	m_stabilizerDeployedFlag : BOOL;
	
	m_sdrivingLeverSensorManualFlag : BOOL;
	
	m_trocarOnFlag :INT;

	m_uiControl : ST_uiControl;
	
	m_joystickValue : vec8d;
	
	m_jntPosReachLimit : vec8b;
	
	m_inMotion : BOOL := false;
END_STRUCT
END_TYPE

// ---- DUTs/Structure/TasksCommunication/ST_CartUIData.TcDUT
TYPE ST_CartUIData :
STRUCT
	m_joystickDataFromUI:ARRAY [0..21] OF USINT;
	m_ctrlEnableFromUI:ST_uiControl;
	m_standColumnHightLimit :LREAL;
	m_surgicalSite : UINT;
	m_surgicalLocation : UINT;
	m_cartDrapingState : UINT;
	m_cartDockingState : UINT;
	m_cartSpecificPosDocking : Vec8d;
	m_cartSpecificPosDraping : Vec8d;
END_STRUCT
END_TYPE

// ---- DUTs/Structure/TasksCommunication/ST_SetupStatus.TcDUT
TYPE ST_SetupStatus :
STRUCT
	// state machine
	m_armState:ARRAY[1..g_sArmNum] OF E_SetupArmState:=[g_sArmNum(SetupArmState_Error)];
	
	// current pose of set arm distal end
	m_curEndPose:ARRAY[1..g_sArmNum] OF ST_Frame;
	
	// position of remote center point
	m_rcPos :ARRAY[1..g_sArmNum] OF Vec3d;
END_STRUCT
END_TYPE

// ---- DUTs/Structure/TasksCommunication/ST_SetupJointData.TcDUT
TYPE ST_SetupJointData :
STRUCT
	// joint position compute with motor encoder
	m_curMotorPos :ARRAY[1..g_sArmNum] OF Vec5d;
	
	// joint position compute with link/abs encoder
	m_curLinkPos :ARRAY[1..g_sArmNum] OF Vec5d;
	
	// target joint position 
	m_cmdJntPos :ARRAY[1..g_sArmNum] OF Vec5d;
	
	// current joint position 
	m_curJntPos :ARRAY[1..g_sArmNum] OF Vec5d;
	
	// current joint position 
	m_curJntVel :ARRAY[1..g_sArmNum] OF Vec5d;
	
	// raw joint current  
	m_rawJntCurrent :ARRAY[1..g_sArmNum] OF Vec5d;
	
	// command joint current 
	m_cmdJntCurrent :ARRAY[1..g_sArmNum] OF Vec5d;
	
END_STRUCT
END_TYPE

// ---- DUTs/Structure/TasksCommunication/ST_SlaveDynaData.TcDUT
TYPE ST_SlaveDynaData :
STRUCT
	// mass matrix in joint space
	m_massMat :ARRAY[1..g_sArmNum] OF Mat3d;
	
	// gravity
	m_gravity :ARRAY[1..g_sArmNum] OF Vec3d;
	
	// instrument out-of-view data
	m_insruViewData :ARRAY[1..g_sArmNum] OF Vec3i;
END_STRUCT
END_TYPE

// ---- DUTs/Structure/TasksCommunication/ST_SlaveUIData.TcDUT
// Output from UI controller
// Input to slave arm control task and cart control task  
TYPE ST_SlaveUIData :
STRUCT
	m_slaveArmDisableFlag :ARRAY[1..4] OF BOOL:=[4(FALSE)];
	m_instruUsageWrite :ARRAY[1..4] OF BOOL:=[4(FALSE)];
	m_armInSelfCheck :  ARRAY [1..g_sArmNum] OF BOOL;
	m_armSelfCheckFinshed :  ARRAY [1..g_sArmNum] OF BOOL;
	m_dumpEnergy : UINT:=51;
END_STRUCT
END_TYPE

// ---- DUTs/Structure/TasksCommunication/ST_MasterJointData.TcDUT
// Output from master arm control task 
// Input to safety task and force controller task
TYPE ST_MasterJointData :
STRUCT
	// joint position compute with motor encoder
	m_curMotorPos :ARRAY[1..g_mArmNum] OF Vec7d;
	
	// joint position compute with link/abs encoder
	m_curLinkPos :ARRAY[1..g_mArmNum] OF Vec7d;
	
	// target joint position 
	m_cmdJntPos :ARRAY[1..g_mArmNum] OF Vec7d;
	
	// current joint position 
	m_curJntPos :ARRAY[1..g_mArmNum] OF Vec7d;
	
	// target joint velocity 
	m_cmdJntVel :ARRAY[1..g_mArmNum] OF Vec7d;
	
	// current joint position 
	m_curJntVel :ARRAY[1..g_mArmNum] OF Vec7d;
	
	// command joint torque 
	m_cmdJntTrq :ARRAY[1..g_mArmNum] OF Vec7d;
	
	// current joint torque 
	m_curJntTrq :ARRAY[1..g_mArmNum] OF Vec7d;
	
	// raw joint current  
	m_rawJntCurrent :ARRAY[1..g_mArmNum] OF Vec7d;
	
	// filtd  joint current  
	m_filtJntCurrent :ARRAY[1..g_mArmNum] OF Vec7d;
	
END_STRUCT
END_TYPE

// ---- DUTs/Structure/TasksCommunication/ST_MotorInputs.TcDUT
TYPE ST_MotorInputs:
STRUCT
	// driver error info
	m_driverError:UDINT;
	
	// driver ethercat status
	m_statusWord:UINT;
	
	// motor/relative encoder from IO
	m_motorEncoder :DINT;
	
	// link/absolute encoder form IO
	m_linkEncoder :DINT;
	
	// motor current from IO
	m_current : DINT;
	
	//motor electrical angle deviation
	m_electriAngleDev : DINT;
	
END_STRUCT
END_TYPE

// ---- DUTs/Structure/TasksCommunication/ST_MotorOutputs.TcDUT
TYPE ST_MotorOutputs :
STRUCT
	// driver control word
	m_controlWord: UINT :=DriverCtrlWord_INIT;
	
	// motor control mode, 0 for position mode, 1 for torque mode
	m_opMode : SINT :=INT_TO_SINT(DriverOPMode_Pos);;
	
	// target motor encoder
	m_cmdMotorEncoder :DINT := 0;
	
	// motor current to IO
	m_cmdCurrent :DINT := 0;
	
	//Powerbox rated current
	m_ratedCurrent:DINT;
END_STRUCT
END_TYPE

// ---- DUTs/Structure/TasksCommunication/ST_SlaveJointData.TcDUT
TYPE ST_SlaveJointData :
STRUCT
	
	// joint position compute with motor encoder
	m_curMotorPos :ARRAY[1..g_sArmNum] OF Vec8d;
	
	// joint position compute with link/abs encoder
	m_curLinkPos :ARRAY[1..g_sArmNum] OF Vec8d;
	
	// target joint position 
	m_cmdJntPos :ARRAY[1..g_sArmNum] OF Vec8d;
	
	// current joint position 
	m_curJntPos :ARRAY[1..g_sArmNum] OF Vec8d;
	
	// current joint position 
	m_curJntVel :ARRAY[1..g_sArmNum] OF Vec8d;
	
	// raw joint current  
	m_rawJntCurrent :ARRAY[1..g_sArmNum] OF Vec8d;
	
	// command joint current 
	m_cmdJntCurrent :ARRAY[1..g_sArmNum] OF Vec8d;
	
	// slave DH joint position 
	m_curDHJntPos :ARRAY[1..g_sArmNum] OF Vec6d;
END_STRUCT
END_TYPE

// ---- DUTs/Structure/TasksCommunication/ST_SafetyData.TcDUT
// Output from safety check task
// Input to master arm control task
TYPE ST_SafetyData :
STRUCT
	m_slaveErrFlag :ARRAY[1..g_sArmNum] OF BOOL :=[4(FALSE)];
	m_setupErrFlag :ARRAY[1..g_sArmNum] OF BOOL :=[4(FALSE)];
	m_cartErrFlag :BOOL :=FALSE;
	m_cartSteadyFootErr :BOOL;
	m_cartWheelErr :BOOL;
	m_cartStandColumnErr :BOOL;
	m_cartAdjustErr :BOOL;
	m_cartOverhangErr :BOOL;
END_STRUCT
END_TYPE

// ---- DUTs/Structure/ST_SlaveArmCtrlCmds.TcDUT
TYPE ST_SlaveArmCtrlCmds :
STRUCT
	// arm control data
	// NOTE: simulated joint position is usd for kinematic controller 
	//		while command joint position is used for real robot controller
	// 		They are identical for the most time, but in some cases, simulated position is filted to get command one 
	m_jntEnableFlag : Vec8i;
	m_jntOPMode : Vec8i;
	m_simJntPos : Vec8d;
	m_cmdJntPos : VEC8d;
	m_cmdJntVel : VEC8d;
	m_cmdJntAcc : VEC8d:=g_zeroVec8d;
	m_cmdJntTrq : VEC8d:=g_zeroVec8d;
	m_cmdCartPose : ST_Frame;
	m_cmdCartTwist : Vec6d;
	m_FFJntTrq :Vec8d:=g_zeroVec8d;
	m_stiffFlag:Vec8i; //---1028
END_STRUCT
END_TYPE

// ---- DUTs/Structure/ST_SlaveInputDataPool.TcDUT
// Struct contains all data from other tasks and controller used for slave control
TYPE ST_SlaveInputDataPool :
STRUCT
		
	// UI information, import from UI controller
	m_UIData :ST_SlaveUIData;
	
	// safety information, import from safety check task
	m_safetyData AT %I*: ST_SafetyData;
	
	// master robot status, copy from MSCommu_MasterStatus
	m_masterStatus :ST_MasterStatus;
	
	// setup arms infromation;
	m_setupStatus AT %I* : ST_SetupStatus;
	
	// slave dynamic data
	m_slaveDynaData AT %I* : ST_SlaveDynaData;
	
END_STRUCT
END_TYPE

// ---- DUTs/Structure/UICommunication/ST_cartOperation.TcDUT
TYPE ST_cartOperation :
STRUCT
	//sterile state ,  0 : unfinshed  , 1 : complete
	m_setupSterileStateArm1 : UINT;
	m_setupSterileStateArm2 : UINT;
	m_setupSterileStateArm3 : UINT;
	m_setupSterileStateArm4 : UINT;
	
	//draping adjust state , 0 : unfinshed  , 1 : finshed
	m_drapingAdjustState : UINT;

	//sterile install state , 0 : unfinshed  , 1 : finshed
	m_setupSterileState : UINT;

	//docking adjust state , 0 : unfinshed  , 1 : finshed
	m_dockingAdjustState : UINT;
	
	//cart in the sterile area 
	m_cartInSterileState : UINT;
	
	//scope installed , 0 : unfinshed  , 1 : finshed
	m_scopeInstalled :UINT;
	
	//robot in surgical allowed , scope installed and an arm mounted instrument
	m_inSurgicalAllowed : UINT;
	
	//arm storage completed
	m_armStorageCompleted : UINT;
END_STRUCT
END_TYPE

// ---- DUTs/Structure/UICommunication/ST_instruInfomation.TcDUT
TYPE ST_instruInfomation :
STRUCT
	//instrument is ready
	m_instruIsConnected : BOOL;
	
	//new instrument  true
	m_newInstrument : BOOL;
	
	//instrument arm in master-slave
	m_instruInMasterSlave : BOOL;
	
	//master send  pedal active
	m_pedalHover : BOOL;
	
	//0 : Passive instrument , 1 : unipolar instrument , 2 : bipolar instrument, 3 : ultrasound knife, 4 : endoscope
	m_instruType : UINT;
	
	//master send  pedal hover
	m_pedalActive : UINT;
	
	//arm id
	m_armId : UINT;
	m_instruID : UINT;
	
	//instrument total number
	m_instruTotalLife : UINT := 100;
	
	//instrument use life (ui write)
	m_useLifeUi : UINT;

	//instrument  use life (plc write)
	m_useLifeplc : UINT;
	
	//instrument serial number
	m_instruSerialNum : LINT;
	
	m_instruPosX : REAL;
	m_instruPosY : REAL;
	m_instruPosZ : REAL;

	//instrument English name 
	m_nameEn : STRING;
	
	//instrument Chinese name 
	m_nameCh : WSTRING;
	
END_STRUCT
END_TYPE

// ---- DUTs/Structure/UICommunication/ST_robotStateMachine.TcDUT
TYPE ST_robotStateMachine :
STRUCT
	m_stateMachineCart : INT;
	m_stateMachineArm1 : INT;
	m_stateMachineArm2 : INT;
	m_stateMachineArm3 : INT;
	m_stateMachineArm4 : INT;

END_STRUCT
END_TYPE

// ---- DUTs/Structure/UICommunication/ST_uiControl.TcDUT
TYPE ST_uiControl :
STRUCT
	//台车自动摆位---姿态调整为建立无菌屏障时所需状态--结束后给定结束信号
	m_drapingEnable : BOOL;
	
	//台车自动摆位---姿态调整为进入无菌区时所需状态（器械对接姿态）--结束后给定结束信号
	m_dockingEnable : BOOL;
	
	//所有机械臂收纳使能
	m_packageEnable : BOOL;
	
	//通过手柄按钮，任意拖动机械臂所有关节
	m_joystickEnable : BOOL;
	
	//相机界面中的使能按钮
	m_cameraJoystickEnable : BOOL;
	
	 //限制高度调整，true:使能，false:禁止
	m_heightLimitAdjustEnable : BOOL;
END_STRUCT
END_TYPE

// ---- DUTs/Type/Mat23.TcDUT
TYPE Mat23 : ARRAY[1..2, 1..3] OF LREAL; END_TYPE

// ---- DUTs/Type/Mat2d.TcDUT
TYPE Mat2d : ARRAY[1..2, 1..2] OF LREAL; END_TYPE

// ---- DUTs/Type/Mat32.TcDUT
TYPE Mat32 : ARRAY[1..3, 1..2] OF LREAL; END_TYPE

// ---- DUTs/Type/Mat53.TcDUT
TYPE Mat53 : ARRAY[1..5, 1..3] OF LREAL; END_TYPE

// ---- DUTs/Type/Mat35.TcDUT
TYPE Mat35 : ARRAY[1..3, 1..5] OF LREAL; END_TYPE

// ---- DUTs/Type/Vec13d.TcDUT
TYPE Vec13d : ARRAY[1..13] OF LREAL; END_TYPE

// ---- DUTs/Type/Vec13di.TcDUT
TYPE Vec13di : ARRAY[1..13] OF DINT; END_TYPE

// ---- DUTs/Type/Vec2d.TcDUT
TYPE Vec2d : ARRAY[1..2] OF LREAL; END_TYPE

// ---- DUTs/Type/Vec2i.TcDUT
TYPE Vec2i : ARRAY[1..2] OF INT; END_TYPE

// ---- DUTs/Type/Vec3i.TcDUT
TYPE Vec3i : ARRAY[1..3] OF INT; END_TYPE

// ---- DUTs/Type/Vec4b.TcDUT
TYPE Vec4b : ARRAY[1..4] OF BOOL; END_TYPE

// ---- DUTs/Type/Vec6b.TcDUT
TYPE Vec6b : ARRAY[1..6] OF BOOL; END_TYPE

// ---- DUTs/Type/Vec8b.TcDUT
TYPE Vec8b : ARRAY[1..8] OF BOOL; END_TYPE

// ---- DUTs/Type/Vec8di.TcDUT
TYPE Vec8di : ARRAY[1..8] OF DINT; END_TYPE

// ---- DUTs/Type/Vec8i.TcDUT
TYPE Vec8i : ARRAY[1..8] OF INT; END_TYPE

// ---- DUTs/Enum/E_DriverCtrlWord.TcDUT
TYPE E_DriverCtrlWord :
(
	DriverCtrlWord_INIT := 6,
	DriverCtrlWord_PREOP := 7,
	DriverCtrlWord_OP := 15,
	DriverCtrlWord_FaultReset := 16#8F
);
END_TYPE

// ---- DUTs/Enum/E_DriverOPMode.TcDUT
TYPE E_DriverOPMode :
(
	DriverOPMode_Pos := 0, // driver position control
	DriverOPMode_Trq :=1, // driver torque control, robot force control
	DriverOPMode_PosTrq :=2, // driver torque control, robot position contorl
	DriverOPMode_Vel :=3, // driver Velocity control
	DriverOPMode_MZPos :=4, //mingzhi driver Position control
	DriverOPMode_cspMZ :=8, //mingzhi driver Sync cycle position mode control
	DriverOPMode_csvMZ :=9 //mingzhi driver Sync cycle position mode control
);
END_TYPE

// ---- DUTs/Enum/E_DriverStatusWord.TcDUT
TYPE E_DriverStatusWord :
(
	DriverStatusWord_INIT := 4641,
	DriverStatusWord_PREOP := 4659,
	DriverStatusWord_OP := 4663,
	
	MZDriverStatusWord_SwitchOnDisable := 16#40,
	MZDriverStatusWord_ReadyToSwitchOn := 16#21,
	MZDriverStatusWord_SwitchOn := 16#33,
	MZDriverStatusWord_OperationEnbale := 16#37,
	MZDriverStatusWord_Fault := 16#08
);
END_TYPE

// ---- SafetyCheck/ErrRecord/checkDelay.TcDUT
TYPE checkDelay  :
STRUCT
	T_armJntEncErr:ARRAY [1..13] OF FB_TON;
	T_driveErr:ARRAY [1..13] OF FB_TON;
	T_linkEncErr:ARRAY [1..13] OF FB_TON;
	T_jntStatusErr:ARRAY [1..13] OF FB_TON;
	T_currentIsNotUpdate:ARRAY [1..13] OF FB_TON;
	T_outOfLimit:ARRAY [1..13] OF FB_TON;
	T_armJntFollowErr:ARRAY [1..13] OF FB_TON;
	T_jntVelErr:ARRAY [1..13] OF FB_TON;
	T_jntCurrentErr:ARRAY [1..13] OF FB_TON;
	T_fixedPointErr:FB_TON;
	T_spacePoseErr:ARRAY [1..13] OF FB_TON;
	T_jntCmdSalta:ARRAY [1..13] OF FB_TON;
	
	T_cartJntEncErr:ARRAY [1..8] OF FB_TON;
	T_cartDriveErr:ARRAY [1..8] OF FB_TON;
	T_cartLinkEncErr:ARRAY [1..8] OF FB_TON;
	T_cartJntStatusErr:ARRAY [1..8] OF FB_TON;
	T_cartCurrentIsNotUpdate:ARRAY [1..8] OF FB_TON;
	T_cartOutOfLimit:ARRAY [1..8] OF FB_TON;
	T_cartJntFollowErr:ARRAY [1..8] OF FB_TON;
	T_cartJntVelErr:ARRAY [1..8] OF FB_TON;
	T_cartJntCurrentErr:ARRAY [1..8] OF FB_TON;
	T_CarMingzhiDriveErr:ARRAY [1..8] OF FB_TON;
END_STRUCT
END_TYPE

// ---- SafetyCheck/ErrRecord/checkDelayTime.TcDUT
TYPE checkDelayTime :
STRUCT
	//motor encoder and joint encoder deviation delay time
	Ti_armJntEncErr:TIME:=T#0.1S;
	//drive error delay time
	Ti_driveErr:TIME:=T#0.1S;
	//joint encoder ununuited delay time
	Ti_linkEncErr:TIME:=T#5S;
	//joint status error delay time 
	Ti_jntStatusErr:TIME:=T#1S;
	//motor current is not update delay time
	Ti_currentIsNotUpdate:TIME:=T#20S;
	//joint postion out of limit
	Ti_outOfLimit:TIME:=T#0.1S;
	//joint follow error delay time
	Ti_armJntFollowErr:TIME:=T#0.1S;
	//joint vel error delay time
	Ti_jntVelErr:TIME:=T#0.05S;
	//joint current error  delay time
	Ti_jntCurrentErr:TIME:=T#0.1S;
	//fixed point postion change of  master-slave state 
	Ti_fixedPointErr:TIME:=T#0.1S;
	//space pose error  delay time
	Ti_spacePoseErr:TIME:=T#0.1S;
	//commend joint position saltation delay time
	Ti_jntCmdSaltationErr:TIME:=T#0.002S;

	
	Ti_CarDualEncDev:TIME:=T#0.02S;
	Ti_CarDriveErr:TIME:=T#1S;
	Ti_CarActSec:TIME:=T#10S;
	Ti_CarJntStatus:TIME:=T#1S;
	Ti_CarTorMotor:TIME:=T#20S;
	Ti_CaroutofLimit:TIME:=T#0.1S;
	Ti_CarFollowDev:TIME:=T#0.02S;
	Ti_CarJntVel:TIME:=T#0.05S;
	Ti_CarJntCurrent:TIME:=T#1S;
	Ti_CarMZDriveErr:TIME:=T#1S;
END_STRUCT
END_TYPE

// ---- SafetyCheck/ErrRecord/checkInputVariable.TcDUT
TYPE checkInputVariable :
STRUCT
	EmergencyStop:BOOL;
	m_cartDriverInput :ARRAY[1..g_cartJntNum] OF ST_MotorInputs; 
	m_cartDriverOutput :ARRAY[1..g_cartJntNum] OF ST_MotorOutputs;
	m_slaveDriverInput :ARRAY[1..g_sJntNum] OF ST_MotorInputs; 
	m_slaveDriverOutput :ARRAY[1..g_sJntNum] OF ST_MotorOutputs;
	m_setupDriverInput :ARRAY[1..g_setupJntNum] OF ST_MotorInputs; 
	m_setupDriverOutput :ARRAY[1..g_setupJntNum] OF ST_MotorOutputs;
	
	m_motorEncoderSaltaValue :  vec13d;  
	m_EtherCATState:ARRAY [1..g_maxArmJoint] OF ST_EtherCATState;		
	m_rcpCheck : BOOL;
	m_spacePoseErr : vec6d;				
	m_cmdArmPos : 	vec6d;		
	m_instruOpenAngle:LREAL;		
	
	m_promptStatus:ARRAY [1..30] OF BOOL;
	m_promptLocation:ARRAY [1..30] OF UDINT;
	
	
	SlaveStopButton:BOOL;
	PCStopButton :UINT;
	MasterStopButton :BOOL;
	
	m_cartEtherCATState:ARRAY [1..g_maxCartJoint] OF ST_EtherCATState;
END_STRUCT
END_TYPE

// ---- SafetyCheck/ErrRecord/checkPermit.TcDUT
TYPE checkPermit :
STRUCT
	m_armJntEncErr :ARRAY [1..13] OF BOOL;
	m_driveErr :ARRAY [1..13] OF BOOL;
	m_jntStatusErr :ARRAY [1..13] OF BOOL;
	m_currentIsNotUpdate :ARRAY [1..13] OF BOOL;
	m_linkEncErr :ARRAY [1..13] OF BOOL;
	m_motPhieErr:ARRAY [1..13] OF BOOL;
	m_outOfLimit :ARRAY [1..13] OF BOOL;
	m_armJntFollowErr :ARRAY [1..13] OF BOOL;
	m_jntVelErr :ARRAY [1..13] OF BOOL;
	m_jntCurrentErr :ARRAY [1..13] OF BOOL;
	m_jntCurrentCtrlErr :ARRAY [1..13] OF BOOL;
	m_fixedPointErr :BOOL;
	m_cmdJntSaltation:ARRAY [1..13] OF BOOL;
	m_spacePoseErr:ARRAY [1..6] OF BOOL;
	m_instruOpenAngle:BOOL;
	

	m_cartJntStatus : vec8b:=[8(TRUE)];
	m_cartCurrentIsNotUpdate : vec8b:=[5(FALSE),3(TRUE)];
	m_cartLinkEncErr : vec8b:=[4(FALSE),4(TRUE)];
	m_cartDriveErr : vec8b:=[8(TRUE)];
	m_cartJntEncErr : vec8b:=[4(FALSE),4(TRUE)];
	m_cartOutOfLimit : vec8b:=[4(FALSE),4(TRUE)];
	m_cartFollowErr : vec8b:=[4(FALSE),4(TRUE)];
	m_cartJntVelErr : vec8b:=[4(FALSE),4(TRUE)];
	m_cartJntCurrentErr : vec8b:=[8(FALSE)];
	m_cartMZDriveErr : vec8b:=[FALSE,FALSE,TRUE,TRUE,TRUE,FALSE,FALSE,FALSE];
END_STRUCT
END_TYPE

// ---- SafetyCheck/ErrRecord/ST_Buffer.TcDUT
TYPE ST_Buffer :
STRUCT
	bFull 		: BOOL;
	sPath		: STRING;
	aBuffer 	: ARRAY[0..MAX_CSV_ROWS ] OF ARRAY [0..MAX_CSV_COLUMNS] OF STRING(MAX_CSV_FIELD_LENGTH) ;
	bBuffer 	: ARRAY[0..MAX_CSV_ROWS ] OF ARRAY [0..MAX_CSV_COLUMNS] OF STRING(MAX_CSV_FIELD_LENGTH) ;
	fbWriter 	: FB_Writer;
END_STRUCT
END_TYPE

// ---- SafetyCheck/ErrRecord/T_Buffer.TcDUT
TYPE T_Buffer: ARRAY[ 0..MAX_CSV_ROWS ] OF ARRAY [0..MAX_CSV_COLUMNS] OF STRING(MAX_CSV_FIELD_LENGTH); (* [] (* TODESC *) *)
END_TYPE

// ---- GVLs/CartJoints/GVL_CartControlParameters.TcGVL
{attribute 'global_init_slot' := '49991'} 
{attribute 'qualified_only'}
VAR_GLOBAL
	// filter cut-off frequency for velocity and torque
	g_curJntVelLpfCutoffFreq :LREAL := 30;
	g_cmdJntTrqLpfCutoffFreq :LREAL := 300;
	g_curJntTrqLpfCutoffFreq :LREAL := 300;
	
	g_curBeamStretchJntInitPos :LREAL := 0.972;
	g_maxCartVel :ARRAY [1..4] OF LREAL:= [0.014, 0.05, 0.05, 0.05];
	
	g_maxJntVel :ARRAY [1..8] OF LREAL:=[0.0025, 0.0025, 2.3, 2.3, 0.014, 5*g_deg2Rad, 0.050, 5*g_deg2Rad];
	g_maxJntAcc :ARRAY [1..8] OF LREAL:=[0.0025*2, 0.0025*2, 2.3*2, 2.3*2, 0.014*2, 5*g_deg2Rad*1.5, 0.050*1.5, 5*g_deg2Rad*1.5];
	
	g_surgicalOrientPos : ARRAY [1..5, 1..3, 1..4]  OF LREAL := [
		0.1, 0.10, 0.10, 0.10,    0.1, -0.10, 0.10, -0.10,	0.1, 0.10, 0.10, -0.10,
		0.2, 0.20, 0.20, 0.20,    0.2, -0.20, 0.20, -0.20,	0.2, 0.20, 0.20, -0.20,
		0.3, 0.25, 0.30, 0.30,    0.3, -0.25, 0.30, -0.30,	0.3, 0.25, 0.30, -0.30,
		0.4, 0.30, 0.35, 0.35,    0.4, -0.30, 0.35, -0.35,	0.4, 0.30, 0.35, -0.35,
		0.5, 0.35, 0.40, 0.40,    0.5, -0.35, 0.40, -0.40,	0.4, 0.30, 0.35, -0.35];
	
	g_surgicalDrapingPos : ARRAY[1..8] OF LREAL := [0, 0, 0, 0, 0.3, 0, 0.2, 0];
	
	g_jntCtrlAngTolHigh :LREAL :=1*g_deg2Rad;
	
	g_cartInitialHeight : UINT := 1805;
	g_cartOpenHorizonLaserHeight : UINT := 1950;
END_VAR

// ---- GVLs/CartJoints/GVL_CartJointEncoderCaliData.TcGVL
{attribute 'qualified_only'}
// Robot5 --joints parameters of setup arms
VAR_GLOBAL
	// absolute encoder value at minimal joint positon
	g_minLinkEncoder :ARRAY[1..g_cartJntNum] OF DINT :=[0, 0, 0, 0, 12912698, 863216, 13187303, 654894];
		 
	// absolute encoder value at maximum joint positon
	g_maxLinkEncoder :ARRAY[1..g_cartJntNum] OF DINT :=[0, 0, 0, 0, 10127418, 3841586, 15255509,16569304 ];
	
	// absolute encoder value at calibrated positon
	g_caliLinkEncoder :ARRAY[1..g_cartJntNum] OF DINT :=[0, 0, 0, 0, 12912698, 2352401, 15255509, 8612099];
	
	 // if absolute encoder value cross zeros within joint motion range
	g_linkEncZeroCross :ARRAY[1..g_cartJntNum] OF INT :=[0, 0, 0, 0, 0, 0, 0, 1];
		 

	// abolute encoder expanded limit buffer in case there is calibrtion error at limit position
	g_linkEncLimitBuffer : DINT := 100000;

	// absolute encoder direction
	g_asbEncoderDir :ARRAY[1..g_cartJntNum] OF INT :=[1, 1, 1, 1, -1, 1, -1, -1];
													
	// flag if joint can rotate multiple cycles
	g_multipleCyclesJoint :ARRAY[1..g_cartJntNum] OF INT :=[0, 0, 0, 0, 0, 0, 0, 0];
		 
	// joint position at link encoder calibrated point
	g_linkEncCaliJntPos :ARRAY[1..g_cartJntNum] OF LREAL :=[0.0, 0.0, 0.0, 0.0, 0.0, 0.0, 0, 0.0];
	
	 // joint SDO address
	g_slaveCartNetID: T_AmsNetId:='169.254.186.39.7.1';
	g_slaveCartJointNetPort:ARRAY[1..g_cartJntNum] OF UINT :=[1005,	1004,	1003,	1002,	1001,   1006,  1007,  1008];

END_VAR

// ---- GVLs/CartJoints/GVL_CartMotorParameters.TcGVL
{attribute 'global_init_slot' := '49991'}
{attribute 'qualified_only'}
VAR_GLOBAL CONSTANT
	// encoder resolution
	//TODO: resolution of joint 2/3 need verification
	g_incEncoderRes :ARRAY[1..g_cartJntNum] OF DINT :=[2(65536), 4*2500, 4*2500, 4*2500, 3(65536)];
	g_absEncoderRes :ARRAY[1..g_cartJntNum] OF DINT :=[1, 1, 1, 1, 8192, 16777215, 8192,16777215];
	
	// reduction ratio
	g_motorReduction :ARRAY[1..g_cartJntNum] OF LREAL :=
		[100.75*2*pi/0.002, 100.75*2*pi/0.002, 160, 160, 
		 5*(2*pi)/0.005, 676.0/49*356, 299.0/14*(2*pi)/0.020, 676.0/49*238];
	g_absEncoderReduction :ARRAY[1..g_cartJntNum] OF LREAL :=[4(1.0), 2*pi/0.002 , 1.0, 2*pi/0.002, 1.0];
	 
	// motor parameters
	g_motorTrqConst :ARRAY[1..g_cartJntNum] OF LREAL :=[ 0.0256, 0.0256, 0.058,0.058,  0.123,0.0292,0.0292,0.0292];
	g_motorMaxCurrent :ARRAY[1..g_cartJntNum] OF LREAL :=[ 41200,41200,50000,50000,  33000,41200,41200,41200];//mA
	
	// motor and absEncoder direction
	g_motorDir :ARRAY[1..g_cartJntNum] OF INT :=[1, 1, 1, 1, 1, 1, -1, -1];
																												 
	// joint position limit
	g_minJntPos: vec8d:=[0, 0, 1, 1, 0, -30*g_deg2Rad, 0.002, -160*g_deg2Rad];	
	g_maxJntPos: vec8d:=[0.053, 0.053, 1, 1,  0.69, 30*g_deg2Rad, 0.498, 160*g_deg2Rad];	
	
	// joint velocity limit
	g_maxJntVel :ARRAY[1..g_cartJntNum] OF LREAL :=[0.0025, 0.0025, 2.3, 2.3, 0.016, 5*g_deg2Rad, 0.050, 5*g_deg2Rad];
	g_maxJntAcc :ARRAY[1..g_cartJntNum] OF LREAL :=[0.0025 * 2, 0.0025 * 2, 2.3 * 2, 2.3 * 2, 0.016 * 2, 5*g_deg2Rad * 2, 0.050 * 2, 5*g_deg2Rad * 2];
END_VAR

// ---- GVLs/configs/robot3/GVL_CartJointEncoderCaliData_3.TcGVL
{attribute 'qualified_only'}
// Robot3 --joints parameters of setup arms
VAR_GLOBAL
	// absolute encoder value at minimal joint positon  2873378  289000
	g_minLinkEncoder :ARRAY[1..g_cartJntNum] OF DINT :=[0, 0, 0, 0, 7300795, 289000, 12042093, 639816];
		 
	// absolute encoder value at maximum joint positon
	g_maxLinkEncoder :ARRAY[1..g_cartJntNum] OF DINT :=[0, 0, 0, 0, 2785280, 2873378, 14110299,2073428 ];
	
	// absolute encoder value at calibrated positon
	g_caliLinkEncoder :ARRAY[1..g_cartJntNum] OF DINT :=[0, 0, 0, 0, 7300795, 1581189, 14110299, 9731340];
	
	 // if absolute encoder value cross zeros within joint motion range
	g_linkEncZeroCross :ARRAY[1..g_cartJntNum] OF INT :=[0, 0, 0, 0, 0, 0, 0, 1];
		 

	// abolute encoder expanded limit buffer in case there is calibrtion error at limit position
	g_linkEncLimitBuffer : DINT := 100000;

	// absolute encoder direction
	g_asbEncoderDir :ARRAY[1..g_cartJntNum] OF INT :=[1, 1, 1, 1, -1, 1, -1, -1];
													
	// flag if joint can rotate multiple cycles
	g_multipleCyclesJoint :ARRAY[1..g_cartJntNum] OF INT :=[0, 0, 0, 0, 0, 0, 0, 0];
		 
	// joint position at link encoder calibrated point
	g_linkEncCaliJntPos :ARRAY[1..g_cartJntNum] OF LREAL :=[0.0, 0.0, 0.0, 0.0, 0.0, 0.0, 0, 0.0];
	
	 // joint SDO address
	g_slaveCartNetID: T_AmsNetId:='169.254.186.39.7.1';
	g_slaveCartJointNetPort:ARRAY[1..g_cartJntNum] OF UINT :=[1005,	1004,	1003,	1002,	1001,   1006,  1007,  1008];

END_VAR

// ---- GVLs/configs/robot3/GVL_SetupArmDynamics_3.TcGVL
{attribute 'global_init_slot' := '49992'}
{attribute 'qualified_only'}
// Robot3 --dynamic parameters of setup arms
VAR_GLOBAL 
	(* setup joint5 gravity parameters. last 5 parameters are defined in slave arm dynamic
	% graParam=[ 9.8*mx0,...
	%            4.92539*m1 + 4.92539*m2 + 4.92539*m3 + 7.8853*m4 + 7.8853*m5 + 9.70463*mx3 - 9.8*my0 - 1.3639*my3 + 9.8*mz1,...
	%            9.8*m5,...
	%            0.41601*m2 + 0.41601*m3 + 0.0000216012*m4 + 0.0000216012*m5 + 9.8*mx1 - 1.3639*mx3 - 9.70463*my3,...
	%            9.8*mz2 - 9.8*my5 - 9.8*my1 + 9.8*mz3 + 9.8*mz4,...
	%            2.19651*m3 + 2.19651*m4 + 0.00000258969*m5 + 8.64766*mx2 - 4.61063*my2 + 9.8*my4 + 9.8*mz5,...
	%            1.1711*m3 + 1.1711*m4 + 0.00000122416*m5 + 4.61063*mx2 - 9.8*mx4 - 9.8*mx5 + 8.64766*my2]';
	*)				
	//setup joint5 gravity parameters
	g_setupJnt5GravityParam :ARRAY[1..4,1..2] OF REAL := 
	[ 0.0000,   54.4806,
	  0.0196,   61.5623,
	  0.0196,   65.0026,
	  0.0196,   59.3080 ];

	(* setup joint3 gravity parameters
	 graParams = [p1mp2,p3,p4]
	 gravity = p1*q^3 + p2*q^2 + p3^q + p4
	 q(- [q0,q1]*)
 	// setup joint3 gravity parameter
	g_setupJnt3GravityParams :ARRAY[1..4, 1..4] OF LREAL :=
	[13129.9, -3010.8, 300.188, -99.7871,
	 14085.9, -3787.37, 476.955, -104.313,
	  6440.78, -1524.39, 415.869, -117.102,
	 22097.9, -5714.59, 558.077, -104.732];
	 
	(* setup joint3 friction parameters
	 graParams = [p1mp2,p3,p4]
	 friciton = p1*q^3 + p2*q^2 + p3^q + p4
	 q(- [q0,q1]*)
 	// setup joint3 friction parameter
	g_setupJnt3FrictionParams :ARRAY[1..4, 1..4] OF LREAL :=
	[-11173.7, 3888.25, -491.555, 79.4495,
	 -17709.9, 6947.19, -897.825, 94.243,
	 -49343.5, 18899.5, -2449.52, 166.011,
	-11537.6, 3698.16, -380.906, 51.8712];
	
	g_setupJnt3GravityPosRange :ARRAY[1..4, 1..2] OF REAL :=
	[0.0189, 	0.1789,
	 0.0182,    0.1784,
	 0.0189,    0.1789,
	 0.0189,    0.1789];
 	
	// joint gravity offset
	g_setupJntGravityOffset :ARRAY[1..4,1..5] OF REAL := 
	[0, 0, 0, 0,  0,
	 0, 0, 0, 0,  0,
	 0, 0, 0, 0,  0,
	 0, 0, 0, 0,  0];

END_VAR

// ---- GVLs/configs/robot3/GVL_SlaveArmDynamics_3.TcGVL
{attribute 'global_init_slot' := '49992'}
{attribute 'qualified_only'}
// Robot3 --dynamic parameters of slave arms
VAR_GLOBAL CONSTANT
	
	// arm gravity parameters
(*graParam=[ 9.8*m5,...
           0.41601*m2 + 0.41601*m3 + 0.0000216012*m4 + 0.0000216012*m5 + 9.8*mx1 - 1.3639*mx3 - 9.70463*my3,...
           9.8*mz2 - 9.8*my5 - 9.8*my1 + 9.8*mz3 + 9.8*mz4,...
           2.19651*m3 + 2.19651*m4 + 0.00000258969*m5 + 8.64766*mx2 - 4.61063*my2 + 9.8*my4 + 9.8*mz5,...
          1.1711*m3 + 1.1711*m4 + 0.00000122416*m5 + 4.61063*mx2 - 9.8*mx4 - 9.8*mx5 + 8.64766*my2]'
*)				
	// robot No.4
	g_gravityParam :ARRAY[1..4,1..5] OF REAL := 
	[ 7.5951,    1.6336,   -4.2417,    9.4106,    4.7289,
	  7.4741,    3.7472,   -4.4567,   10.5517,    7.6095,
	  7.6732,    3.7472,   -4.4458,    9.6721,    7.2742,
	  7.4582,    3.5688,   -3.7215,    9.2746,    5.7641];
	 
	g_gravityTrocar :ARRAY[1..5] OF REAL :=[0.1661, -0.4124,  0.0964,   -0.7987,   -0.6999 ];
	g_gravityInstrument :ARRAY[1..5] OF REAL :=[ 3.1217,  -0.3099,   0.0778,   -1.2498,   -0.8041];
	g_gravityEndoscope :ARRAY[1..5] OF REAL :=[10.8619,  -0.8575,   -1.0274,   -0.2425,   -0.0869];
	
	// joint friction(with instrument mounted)
	g_slaveJntFriction :ARRAY[1..g_sArmNum, 1..g_sJntNum] OF LREAL :=
			[ 5.3354,    9.5437,    4.6271,  0.03, 0.03, 0.03, 0.03, 0,
			  4.5927,    9.6040,    3.7367, 0.03, 0.03, 0.03, 0,
		      4.3557,    8.4286,    5.9078,  0.03, 0.03, 0.03, 0.03, 0,
              4.1447,    7.2202,    6.8253,  0.03, 0.03, 0.03, 0.03, 0	 ];
			  
	//################ DO NOT modify parameters below ###########################
	//################ dynamic reference model parameters below ###########################
	// link mass [m1, m2, m3, m4, m5]
	g_linkMass :ARRAY[1..5] OF LREAL :=[5.6565, 1.4613, 1.149, 1.5362, 0.6679] ;
	
	// lin center of amss
	g_linkCOM :ARRAY[1..5,1..3] OF LREAL :=  [ 0.0566,    0.0302,   -0.4685,
											   0.1191,   -0.0011,   -0.0588,
											   0.1238,    0.0003,   -0.0120,
											   0.0427,    0.0924,   -0.0004,
											   -0.0262,        0,   -0.0292];
	// link  inertial
    // [Ixx,Iyy,Izz, Ixy,Ixz, Iyz]
 	g_linkInertia :ARRAY[1..5,1..6] OF LREAL :=[0.0735,    0.0738,    0.0144,    0.0016,   -0.0000,   -0.0079,
												0.0016,    0.0190,    0.0185,         0,    0.0027,         0,
											   0.0009,    0.0167,    0.0166,         0,    0.0012,         0,
												0.0009,    0.0167,    0.0166,         0,    0.0012,         0,
											  0.0009,    0.0167,    0.0166,         0,    0.0012,         0];

	
	//  motor inertial at link size
	g_motorInertia :ARRAY[1..3] OF LREAL := [0.00004487, 0.00004487, 0.0000002280];

END_VAR

// ---- GVLs/configs/robot3/GVL_SetupJointEncoderCaliData_3.TcGVL
{attribute 'qualified_only'}
// Robot3 --joints parameters of setup arms
VAR_GLOBAL
	// absolute encoder value at minimal joint positon
	g_minLinkEncoder :ARRAY[1..g_sArmNum, 1..g_setupJntNum] OF DINT :=
		[5813168, 22663264, 1978132, 1938100, 13659124,
		 13487924, 17543781, 3084321, 10238892, 1028618,
		  3186404, 15837168, 878439, 6065586, 9487992,
		  553720, 24385008, 4169014, 6084058, 984346];
		 
	// absolute encoder value at maximum joint positon
	g_maxLinkEncoder :ARRAY[1..g_sArmNum, 1..g_setupJntNum] OF DINT :=
		[1055544, 21209065, 1176866, 385208, 4921448,
		 8781908, 16093586, 2285859, 8654922, 9089506,
		 15289572, 14389054, 85603, 4478314, 767644,
		  12599264, 22936561, 3373290, 4489778, 9055426];
	
	// absolute encoder value at calibrated positon
	g_caliLinkEncoder :ARRAY[1..g_sArmNum, 1..g_setupJntNum] OF DINT :=
		[3511708, 21210622, 1977753, 9295000, 9311970,
		  11205276, 16093586, 3084321, 783598, 13445092,
		 844948, 14389054, 878439, 13364040, 5122582,
		  14940512, 22936561, 4169014, 13457164, 13393096];
	
	 // if absolute encoder value cross zeros within joint motion range
	g_linkEncZeroCross :ARRAY[1..g_sArmNum, 1..g_setupJntNum] OF INT :=
		[0, 0, 0, 1, 0,
		 0, 0, 0, 1, 1,
		 1, 0, 0, 1, 0,
		 1, 0, 0, 1, 1];
		 
//################ DO NOT modify parameters below ###########################
	// abolute encoder expanded limit buffer in case there is calibrtion error at limit position
	g_linkEncLimitBuffer : DINT := 100000;

	// absolute encoder direction
	g_asbEncoderDir :ARRAY[1..g_setupJntNum] OF INT :=[-1, -1, -1, 1, -1];
													
	// flag if joint can rotate multiple cycles
	g_multipleCyclesJoint :ARRAY[1..g_sArmNum, 1..g_setupJntNum] OF INT :=
		[0, 0, 0, 0, 0,
		 0, 0, 0, 0, 0,
		 0, 0, 0, 0, 0,
		 0, 0, 0, 0, 0];
		 
	// joint position at link encoder calibrated point
	g_linkEncCaliJntPos :ARRAY[1..g_sArmNum, 1..g_setupJntNum] OF LREAL :=
		[-140*g_deg2Rad, 0.779, 0.0, 90.0*g_deg2Rad, 0.0,
		 -115*g_deg2Rad, 0.607, 0.0, 90.0*g_deg2Rad, 0.0,
		 -65*g_deg2Rad, 0.607, 0.0, 90.0*g_deg2Rad, 0.0,
 		 -40*g_deg2Rad, 0.779, 0.0, 90.0*g_deg2Rad, 0.0];
	
END_VAR

// ---- GVLs/configs/robot3/GVL_SlaveJointEncoderCaliData_3.TcGVL
{attribute 'qualified_only'}
// Robot3 --joints parameters of slave arms
VAR_GLOBAL CONSTANT	
	// absolute encoder value at minimal joint positon
	g_minLinkEncoder :ARRAY[1..g_sArmNum, 1..g_sJntNum] OF DINT :=
		[796618, 12395160, 5368016, 0, 0, 0, 0, 0,
		 13317378, 3888760, 9175760, 0, 0, 0, 0, 0,
		 823964, 3955316, 15205696, 0, 0, 0, 0, 0,
		 4820816, 7977020, 9226720, 0, 0, 0, 0, 0];
		 
	// absolute encoder value at maximum joint positon
	g_maxLinkEncoder :ARRAY[1..g_sArmNum, 1..g_sJntNum] OF DINT :=
		[15464922, 5123844, 14570432, 0, 0, 0, 0, 0,
		 11230582, 13464106, 1613344, 0, 0, 0, 0, 0,
		 15526052, 13536910, 7701984, 0, 0, 0, 0, 0,
		 2731020, 789080, 1671808, 0, 0, 0, 0, 0];
	
	// absolute encoder value at calibrated positon
	g_caliLinkEncoder :ARRAY[1..g_sArmNum, 1..g_sJntNum] OF DINT :=
		[8162412, 8169482, 14570432, 15377856,15482848, 7058832, 6935120, 7155184,
		 3932766, 16478880, 1613344, 15324752, 15485488, 7135776, 7032592, 6946704,
		 8248074, 16595424, 7701984, 15349408, 15361392, 7017904, 6757296, 7028608,
		 12196142, 3807946, 1671808, 15274368, 15387696, 6812992, 7016768, 7073088];
	
	 // if absolute encoder value cross zeros within joint motion range
	 // NOTICE: joint 7 is always 0.
	g_linkEncZeroCross :ARRAY[1..g_sArmNum, 1..g_sJntNum] OF INT :=
		[0, 0, 0, 1, 1, 1, 1, 1,
		 1, 1, 1, 1, 1, 1, 1, 1,
		 0, 1, 1, 1, 1, 1, 1, 1,
		 1, 0, 1, 1, 1, 1, 1, 1];
		 
	 // joint SDO address
	g_slaveArmNetID: ARRAY[1..4] OF T_AmsNetId:=['169.254.186.39.3.1','169.254.186.39.8.1','169.254.186.39.9.1','169.254.186.39.10.1'];
	g_slaveJointNetPort:ARRAY[1..g_sArmNum,1..g_sJntNum] OF UINT :=[
		1006,	1007,	1008,	2(1009),	3(1010),
		1006,	1007,	1008,	2(1009),	3(1010),
		1006,	1007,	1008,	2(1009),	3(1010),
		1006,	1007,	1008,	2(1009),	3(1010)];
		
//################ DO NOT modify parameters below ###########################
	// abolute encoder expanded limit buffer in case there is calibrtion error at limit position
	g_linkEncLimitBuffer : DINT := 100000;
	
	// absolute encoder direction
	g_asbEncoderDir :ARRAY[1..g_sJntNum] OF INT :=[1, -1, 1, 1, 1, 1, 1, 1];
	
	// flag if joint can rotate multiple cycles
	g_multipleCyclesJoint :ARRAY[1..g_sArmNum, 1..g_sJntNum] OF INT :=
		[0, 0, 0, 1, 1, 1, 1, 1,
		 0, 0, 0, 1, 1, 1, 1, 1,
		 0, 0, 0, 1, 1, 1, 1, 1,
		 0, 0, 0, 1, 1, 1, 1, 1];
		 
	// joint position at link encoder calibrated point
	g_linkEncCaliJntPos :ARRAY[1..g_sJntNum] OF LREAL :=
		[0.0, -PI/2 + 8*g_deg2rad, 0.581633, 5(0.0)];

	
END_VAR

// ---- GVLs/configs/robot5/GVL_CartJointEncoderCaliData_5.TcGVL
{attribute 'qualified_only'}
// Robot5 --joints parameters of setup arms
VAR_GLOBAL
	// absolute encoder value at minimal joint positon
	g_minLinkEncoder :ARRAY[1..g_cartJntNum] OF DINT :=[0, 0, 0, 0, 39509461, 14558528, 57761547, 8171292];
		 
	// absolute encoder value at maximum joint positon
	g_maxLinkEncoder :ARRAY[1..g_cartJntNum] OF DINT :=[0, 0, 0, 0, 36724181, 577308, 59809539,7327520 ];
	
	// absolute encoder value at calibrated positon
	g_caliLinkEncoder :ARRAY[1..g_cartJntNum] OF DINT :=[0, 0, 0, 0, 39509461, 15956526, 59809539, 16172652];
	
	 // if absolute encoder value cross zeros within joint motion range
	g_linkEncZeroCross :ARRAY[1..g_cartJntNum] OF INT :=[0, 0, 0, 0, 0, 1, 0, 1];
		 

	// abolute encoder expanded limit buffer in case there is calibrtion error at limit position
	g_linkEncLimitBuffer : DINT := 100000;

	// absolute encoder direction
	g_asbEncoderDir :ARRAY[1..g_cartJntNum] OF INT :=[1, 1, 1, 1, -1, 1, -1, -1];
													
	// flag if joint can rotate multiple cycles
	g_multipleCyclesJoint :ARRAY[1..g_cartJntNum] OF INT :=[0, 0, 0, 0, 0, 0, 0, 0];
		 
	// joint position at link encoder calibrated point
	g_linkEncCaliJntPos :ARRAY[1..g_cartJntNum] OF LREAL :=[0.0, 0.0, 0.0, 0.0, 0.0, 0.0, 0, 0.0];
	
	 // joint SDO address
	g_slaveCartNetID: T_AmsNetId:='169.254.186.39.7.1';
	g_slaveCartJointNetPort:ARRAY[1..g_cartJntNum] OF UINT :=[1005,	1004,	1003,	1002,	1001,   1006,  1007,  1008];

END_VAR

// ---- GVLs/configs/robot5/GVL_SetupArmDynamics_5.TcGVL
{attribute 'global_init_slot' := '49992'}
{attribute 'qualified_only'}
// Robot5 --dynamic parameters of setup arms
VAR_GLOBAL 
	(* setup joint5 gravity parameters. last 5 parameters are defined in slave arm dynamic
	% graParam=[ 9.8*mx0,...
	%            4.92539*m1 + 4.92539*m2 + 4.92539*m3 + 7.8853*m4 + 7.8853*m5 + 9.70463*mx3 - 9.8*my0 - 1.3639*my3 + 9.8*mz1,...
	%            9.8*m5,...
	%            0.41601*m2 + 0.41601*m3 + 0.0000216012*m4 + 0.0000216012*m5 + 9.8*mx1 - 1.3639*mx3 - 9.70463*my3,...
	%            9.8*mz2 - 9.8*my5 - 9.8*my1 + 9.8*mz3 + 9.8*mz4,...
	%            2.19651*m3 + 2.19651*m4 + 0.00000258969*m5 + 8.64766*mx2 - 4.61063*my2 + 9.8*my4 + 9.8*mz5,...
	%            1.1711*m3 + 1.1711*m4 + 0.00000122416*m5 + 4.61063*mx2 - 9.8*mx4 - 9.8*mx5 + 8.64766*my2]';
	*)				
	//setup joint5 gravity parameters
	g_setupJnt5GravityParam :ARRAY[1..4,1..2] OF REAL := 
	[ 0.0000,   54.4806,
	  0.0196,   61.5623,
	  0.0196,   65.0026,
	  0.0196,   59.3080 ];

	(* setup joint3 gravity parameters
	 graParams = [p1,p2,p3,p4]
	 gravity = p1*q^3 + p2*q^2 + p3^q + p4
	 q(- [q0,q1]*)
 	// setup joint3 gravity parameter
	g_setupJnt3GravityParams :ARRAY[1..4, 1..4] OF LREAL :=
	[17452.1, -4008.76, 401.477, -117.096,
	 8476.95, -1240.58, 104.752, -105.76,
	 14956.5, -4297.99, 622.564, -131.776,
	 14926.3, -2807.93, 154.175, -103.6];
	 
	(* setup joint3 friction parameters
	 graParams = [p1mp2,p3,p4]
	 friciton = p1*q^3 + p2*q^2 + p3^q + p4
	 q(- [q0,q1]*)
 	// setup joint3 friction parameter
	g_setupJnt3FrictionParams :ARRAY[1..4, 1..4] OF LREAL :=
	[ -18790.6, 5987.36, -582.149, 60.6865,
	  -19818.6, 7327.61, -903.65, 81.3597,
	-60054.7, 22353.3, -2711.22, 147.637,
	-25150.3, 8097.23, -822.128, 75.4573];
	
	g_setupJnt3GravityPosRange :ARRAY[1..4, 1..2] OF REAL :=
	[0.0189, 	0.1789,
	 0.0182,    0.1784,
	 0.0189,    0.1789,
	 0.0189,    0.1789];
 	
	 
	// joint gravity offset
	g_setupJntGravityOffset :ARRAY[1..4,1..5] OF REAL := 
	[0, 0, 10, 0,  0,
	 0, 0, 10, 0,  0,
	 0, 0, 10, 0,  0,
	 0, 0, 10, 0,  0];

END_VAR

// ---- GVLs/configs/robot5/GVL_SlaveArmDynamics_5.TcGVL
{attribute 'global_init_slot' := '49992'}
{attribute 'qualified_only'}
// Robot5 --dynamic parameters of slave arms
VAR_GLOBAL CONSTANT
	// arm gravity parameters
(*graParam=[ 9.8*m5,...
           0.41601*m2 + 0.41601*m3 + 0.0000216012*m4 + 0.0000216012*m5 + 9.8*mx1 - 1.3639*mx3 - 9.70463*my3,...
           9.8*mz2 - 9.8*my5 - 9.8*my1 + 9.8*mz3 + 9.8*mz4,...
           2.19651*m3 + 2.19651*m4 + 0.00000258969*m5 + 8.64766*mx2 - 4.61063*my2 + 9.8*my4 + 9.8*mz5,...
          1.1711*m3 + 1.1711*m4 + 0.00000122416*m5 + 4.61063*mx2 - 9.8*mx4 - 9.8*mx5 + 8.64766*my2]'
*)			
	// robot No.4
	g_gravityParam :ARRAY[1..4,1..5] OF REAL := 
	[ 7.5951,    1.6336,   -4.2417,    9.4106,    4.7289,
	  7.4741,    3.7472,   -4.4567,   10.5517,    7.6095,
	  7.6732,    3.7472,   -4.4458,    9.6721,    7.2742,
	  7.4582,    3.5688,   -3.7215,    9.2746,    5.7641];
	 
	g_gravityTrocar :ARRAY[1..5] OF REAL :=[0.1661, -0.4124,  0.0964,   -0.7987,   -0.6999 ];
	g_gravityInstrument :ARRAY[1..5] OF REAL :=[ 3.1217,  -0.3099,   0.0778,   -1.2498,   -0.8041];
	g_gravityEndoscope :ARRAY[1..5] OF REAL :=[10.8619,  -0.8575,   -1.0274,   -0.2425,   -0.0869];
	
	// joint friction(with instrument mounted)
	g_slaveJntFriction :ARRAY[1..g_sArmNum, 1..g_sJntNum] OF LREAL :=
			[ 5.3354,    9.5437,    4.6271,  0.03, 0.03, 0.03, 0.03, 0,
			  4.5927,    9.6040,    3.7367, 0.03, 0.03, 0.03, 0,
		      4.3557,    8.4286,    5.9078,  0.03, 0.03, 0.03, 0.03, 0,
              4.1447,    7.2202,    6.8253,  0.03, 0.03, 0.03, 0.03, 0	 ];
			  
	//################ DO NOT modify parameters below ###########################
	//################ dynamic reference model parameters below ###########################
	// link mass [m1, m2, m3, m4, m5]
	g_linkMass :ARRAY[1..5] OF LREAL :=[5.6565, 1.4613, 1.149, 1.5362, 0.6679] ;
	
	// lin center of amss
	g_linkCOM :ARRAY[1..5,1..3] OF LREAL :=  [ 0.0566,    0.0302,   -0.4685,
											   0.1191,   -0.0011,   -0.0588,
											   0.1238,    0.0003,   -0.0120,
											   0.0427,    0.0924,   -0.0004,
											   -0.0262,        0,   -0.0292];
	// link  inertial
    // [Ixx,Iyy,Izz, Ixy,Ixz, Iyz]
 	g_linkInertia :ARRAY[1..5,1..6] OF LREAL :=[0.0735,    0.0738,    0.0144,    0.0016,   -0.0000,   -0.0079,
												0.0016,    0.0190,    0.0185,         0,    0.0027,         0,
											   0.0009,    0.0167,    0.0166,         0,    0.0012,         0,
												0.0009,    0.0167,    0.0166,         0,    0.0012,         0,
											  0.0009,    0.0167,    0.0166,         0,    0.0012,         0];

	
	//  motor inertial at link size
	g_motorInertia :ARRAY[1..3] OF LREAL := [0.00004487, 0.00004487, 0.0000002280];
	
END_VAR

// ---- GVLs/configs/robot5/GVL_SetupJointEncoderCaliData_5.TcGVL
{attribute 'qualified_only'}
// Robot5 --joints parameters of setup arms
VAR_GLOBAL
	// absolute encoder value at minimal joint positon
	g_minLinkEncoder :ARRAY[1..g_sArmNum, 1..g_setupJntNum] OF DINT :=
		[10820860, 64919092, 57409031, 1851032, 1117696,
		 15040796, 19250150, 52220472, 1865736, 5370968,
		 15165364, 61524935, 56328180, 10224882, 1019944,
		 12364020, 63250814, 55221937, 14440620, 5319980];
		 
	// absolute encoder value at maximum joint positon
	g_maxLinkEncoder :ARRAY[1..g_sArmNum, 1..g_setupJntNum] OF DINT :=
		[6102024, 63534315, 56635702, 394750, 9155824,
		 10329032, 17795974, 51417699, 303438, 13416490,
		 10495464, 60071845, 55514393, 8671968, 9053316,
		 7627212, 61793781, 54433447, 12871432, 13365450];
	
	// absolute encoder value at calibrated positon
	g_caliLinkEncoder :ARRAY[1..g_sArmNum, 1..g_setupJntNum] OF DINT :=
		[8479084, 63534315, 57409031, 9224498, 13527366,
		 12606456, 17795974, 52220472, 9143734, 994974,
		 12863028, 60071845, 56328180, 774190, 13414374,
		 10068792, 61793781, 55221937, 5068940, 951234];
	
	 // if absolute encoder value cross zeros within joint motion range
	g_linkEncZeroCross :ARRAY[1..g_sArmNum, 1..g_setupJntNum] OF INT :=
		[0, 0, 0, 1, 1,
		 0, 0, 0, 1, 1,
		 0, 0, 0, 1, 1,
		 0, 0, 0, 1, 1];
		 
//################ DO NOT modify parameters below ###########################
	// abolute encoder expanded limit buffer in case there is calibrtion error at limit position
	g_linkEncLimitBuffer : DINT := 100000;

	// absolute encoder direction
	g_asbEncoderDir :ARRAY[1..g_setupJntNum] OF INT :=[-1, -1, -1, 1, -1];
													
	// flag if joint can rotate multiple cycles
	g_multipleCyclesJoint :ARRAY[1..g_sArmNum, 1..g_setupJntNum] OF INT :=
		[0, 0, 0, 0, 0,
		 0, 0, 0, 0, 0,
		 0, 0, 0, 0, 0,
		 0, 0, 0, 0, 0];
		 
	// joint position at link encoder calibrated point
	g_linkEncCaliJntPos :ARRAY[1..g_sArmNum, 1..g_setupJntNum] OF LREAL :=
		[-140*g_deg2Rad, 0.779, 0.0, 90.0*g_deg2Rad, 0.0,
		 -115*g_deg2Rad, 0.607, 0.0, 90.0*g_deg2Rad, 0.0,
		 -65*g_deg2Rad, 0.607, 0.0, 90.0*g_deg2Rad, 0.0,
 		 -40*g_deg2Rad, 0.779, 0.0, 90.0*g_deg2Rad, 0.0];
	

END_VAR

// ---- GVLs/configs/robot5/GVL_SlaveJointEncoderCaliData_5.TcGVL
{attribute 'qualified_only'}
// Robot5 --joints parameters of slave arms
VAR_GLOBAL CONSTANT
	// absolute encoder value at minimal joint positon
	g_minLinkEncoder :ARRAY[1..g_sArmNum, 1..g_sJntNum] OF DINT :=
		[13299286, 12259316, 8131200, 0, 0, 0, 0, 0,
		 7690928, 8194684, 1783424, 0, 0, 0, 0, 0,
		 13300276, 12243976, 15232032, 0, 0, 0, 0, 0,
		 752828, 16341268, 3536512, 0, 0, 0, 0, 0];
		 
	// absolute encoder value at maximum joint positon
	g_maxLinkEncoder :ARRAY[1..g_sArmNum, 1..g_sJntNum] OF DINT :=
		[11218724, 5032692, 509984, 0, 0, 0, 0, 0,
		 15388748, 943300, 10993024, 0, 0, 0, 0, 0,
		 11204586, 5012744, 7690928, 0, 0, 0, 0, 0,
		 15415998, 9127988, 12720912, 0, 0, 0, 0, 0];
	
	// absolute encoder value at calibrated positon
	g_caliLinkEncoder :ARRAY[1..g_sArmNum, 1..g_sJntNum] OF DINT :=
		[3882398, 8083626, 509984, 13079328, 101984, 14934512, 4402512, 5578752,
		 8049042, 3955388, 10993024, 15376976, 15429216, 6997360, 7093456, 7154688,
		 3865836, 8052426, 7690928, 15280848, 15470720, 7024336, 7061984, 7187520,
		 8117082, 12176494, 12720912, 15362624, 15350880, 6971776, 6970208, 7079008];
	
	 // if absolute encoder value cross zeros within joint motion range
	 // NOTICE: joint 7 is always 0.
	g_linkEncZeroCross :ARRAY[1..g_sArmNum, 1..g_sJntNum] OF INT :=
		[1, 0, 1, 1, 1, 1, 1, 1,
		 0, 0, 0, 1, 1, 1, 1, 1,
		 1, 0, 1, 1, 1, 1, 1, 1,
		 0, 0, 0, 1, 1, 1, 1, 1];
		 
	 // joint SDO address
	g_slaveArmNetID: ARRAY[1..4] OF T_AmsNetId:=['169.254.186.39.3.1','169.254.186.39.8.1','169.254.186.39.9.1','169.254.186.39.10.1'];
	g_slaveJointNetPort:ARRAY[1..g_sArmNum,1..g_sJntNum] OF UINT :=[
		1006,	1007,	1008,	2(1009),	3(1010),
		1006,	1007,	1008,	2(1009),	3(1010),
		1006,	1007,	1008,	2(1009),	3(1010),
		1006,	1007,	1008,	2(1009),	3(1010)];
		
//################ DO NOT modify parameters below ###########################
	// abolute encoder expanded limit buffer in case there is calibrtion error at limit position
	g_linkEncLimitBuffer : DINT := 100000;
	
	// absolute encoder direction
	g_asbEncoderDir :ARRAY[1..g_sJntNum] OF INT :=[1, -1, 1, 1, 1, 1, 1, 1];
	
	// flag if joint can rotate multiple cycles
	g_multipleCyclesJoint :ARRAY[1..g_sArmNum, 1..g_sJntNum] OF INT :=
		[0, 0, 0, 1, 1, 1, 1, 1,
		 0, 0, 0, 1, 1, 1, 1, 1,
		 0, 0, 0, 1, 1, 1, 1, 1,
		 0, 0, 0, 1, 1, 1, 1, 1];
		 
	// joint position at link encoder calibrated point
	g_linkEncCaliJntPos :ARRAY[1..g_sJntNum] OF LREAL :=
		[0.0, -PI/2 + 8*g_deg2rad, 0.581633, 5(0.0)];

	
END_VAR

// ---- GVLs/configs/robot4/GVL_SetupArmDynamics_4.TcGVL
{attribute 'global_init_slot' := '49992'}
{attribute 'qualified_only'}
// Robot4 --dynamic parameters of setup arms
VAR_GLOBAL 
	(* setup joint5 gravity parameters. last 5 parameters are defined in slave arm dynamic
	% graParam=[ 9.8*mx0,...
	%            4.92539*m1 + 4.92539*m2 + 4.92539*m3 + 7.8853*m4 + 7.8853*m5 + 9.70463*mx3 - 9.8*my0 - 1.3639*my3 + 9.8*mz1,...
	%            9.8*m5,...
	%            0.41601*m2 + 0.41601*m3 + 0.0000216012*m4 + 0.0000216012*m5 + 9.8*mx1 - 1.3639*mx3 - 9.70463*my3,...
	%            9.8*mz2 - 9.8*my5 - 9.8*my1 + 9.8*mz3 + 9.8*mz4,...
	%            2.19651*m3 + 2.19651*m4 + 0.00000258969*m5 + 8.64766*mx2 - 4.61063*my2 + 9.8*my4 + 9.8*mz5,...
	%            1.1711*m3 + 1.1711*m4 + 0.00000122416*m5 + 4.61063*mx2 - 9.8*mx4 - 9.8*mx5 + 8.64766*my2]';
	*)				
	//setup joint5 gravity parameters
	g_setupJnt5GravityParam :ARRAY[1..4,1..2] OF REAL := 
	[ 0.0000,   54.4806,
	  0.0196,   61.5623,
	  0.0196,   65.0026,
	  0.0196,   59.3080 ];

	(* setup joint3 gravity parameters
	 graParams = [p1,p2,p3,p4]
	 gravity = p1*q^3 + p2*q^2 + p3^q + p4
	 q(- [q0,q1]*)
 	// setup joint3 gravity parameter
	g_setupJnt3GravityParams :ARRAY[1..4, 1..4] OF LREAL :=
	[ 12732.1, -2686.58, 277.075, -95.1403,
	 -4213.4, 1194.4, 207.745, -118.926,
	3798.81, -862.596, 397.288, -127.846,
	 35991.5, -10457.4, 1058.33, -122.463];
	 
	(* setup joint3 friction parameters
	 graParams = [p1mp2,p3,p4]
	 friciton = p1*q^3 + p2*q^2 + p3^q + p4
	 q(- [q0,q1]*)
 	// setup joint3 friction parameter
	g_setupJnt3FrictionParams :ARRAY[1..4, 1..4] OF LREAL :=
	[  -41668.6, 14453.2, -1563.43, 100.562,
	 -16563.6, 8089.53, -1307.53, 112.977,
	-39448.5, 15129.4, -1976.17, 137.28,
	-26846.1, 9145.03, -1006.01, 79.1108];
	
	g_setupJnt3GravityPosRange :ARRAY[1..4, 1..2] OF REAL :=
	[ 0.0189,    0.1788,
	  0.0189,    0.1790,
	  0.0188,    0.1788,
	  0.0188,    0.1788];
 	
	 
	// joint gravity offset
	g_setupJntGravityOffset :ARRAY[1..4,1..5] OF REAL := 
	[0, 0, 0, 0,  0,
	 0, 0, 0, 0,  0,
	 0, 0, 0, 0,  0,
	 0, 0, 0, 0,  0];

END_VAR

// ---- GVLs/configs/robot4/GVL_SlaveArmDynamics_4.TcGVL
{attribute 'global_init_slot' := '49992'}
{attribute 'qualified_only'}
// Robot4 --dynamic parameters of slave arms
VAR_GLOBAL CONSTANT
	
	// arm gravity parameters
(*graParam=[ 9.8*m5,...
           0.41601*m2 + 0.41601*m3 + 0.0000216012*m4 + 0.0000216012*m5 + 9.8*mx1 - 1.3639*mx3 - 9.70463*my3,...
           9.8*mz2 - 9.8*my5 - 9.8*my1 + 9.8*mz3 + 9.8*mz4,...
           2.19651*m3 + 2.19651*m4 + 0.00000258969*m5 + 8.64766*mx2 - 4.61063*my2 + 9.8*my4 + 9.8*mz5,...
          1.1711*m3 + 1.1711*m4 + 0.00000122416*m5 + 4.61063*mx2 - 9.8*mx4 - 9.8*mx5 + 8.64766*my2]'
*)			
	// robot No.4
	g_gravityParam :ARRAY[1..4,1..5] OF REAL := 
	[ 7.5951,    1.6336,   -4.2417,    9.4106,    4.7289,
	  7.4741,    3.7472,   -4.4567,   10.5517,    7.6095,
	  7.6732,    3.7472,   -4.4458,    9.6721,    7.2742,
	  7.4582,    3.5688,   -3.7215,    9.2746,    5.7641];
	 
	g_gravityTrocar :ARRAY[1..5] OF REAL :=[0.1661, -0.4124,  0.0964,   -0.7987,   -0.6999 ];
	g_gravityInstrument :ARRAY[1..5] OF REAL :=[ 3.1217,  -0.3099,   0.0778,   -1.2498,   -0.8041];
	g_gravityEndoscope :ARRAY[1..5] OF REAL :=[10.8619,  -0.8575,   -1.0274,   -0.2425,   -0.0869];
	
	// joint friction(with instrument mounted)
	g_slaveJntFriction :ARRAY[1..g_sArmNum, 1..g_sJntNum] OF LREAL :=
			[ 5.3354,    9.5437,    4.6271,  0.03, 0.03, 0.03, 0.03, 0,
			  4.5927,    9.6040,    3.7367, 0.03, 0.03, 0.03, 0,
		      4.3557,    8.4286,    5.9078,  0.03, 0.03, 0.03, 0.03, 0,
              4.1447,    7.2202,    6.8253,  0.03, 0.03, 0.03, 0.03, 0	 ];
			  
	//################ DO NOT modify parameters below ###########################
	//################ dynamic reference model parameters below ###########################
	// link mass [m1, m2, m3, m4, m5]
	g_linkMass :ARRAY[1..5] OF LREAL :=[5.6565, 1.4613, 1.149, 1.5362, 0.6679] ;
	
	// lin center of amss
	g_linkCOM :ARRAY[1..5,1..3] OF LREAL :=  [ 0.0566,    0.0302,   -0.4685,
											   0.1191,   -0.0011,   -0.0588,
											   0.1238,    0.0003,   -0.0120,
											   0.0427,    0.0924,   -0.0004,
											   -0.0262,        0,   -0.0292];
	// link  inertial
    // [Ixx,Iyy,Izz, Ixy,Ixz, Iyz]
 	g_linkInertia :ARRAY[1..5,1..6] OF LREAL :=[0.0735,    0.0738,    0.0144,    0.0016,   -0.0000,   -0.0079,
												0.0016,    0.0190,    0.0185,         0,    0.0027,         0,
											   0.0009,    0.0167,    0.0166,         0,    0.0012,         0,
												0.0009,    0.0167,    0.0166,         0,    0.0012,         0,
											  0.0009,    0.0167,    0.0166,         0,    0.0012,         0];

	
	//  motor inertial at link size
	g_motorInertia :ARRAY[1..3] OF LREAL := [0.00004487, 0.00004487, 0.0000002280];
	
END_VAR

// ---- GVLs/configs/robot4/GVL_SlaveJointEncoderCaliData_4.TcGVL
{attribute 'qualified_only'}
// Robot4 --joints parameters of slave arms
VAR_GLOBAL CONSTANT
	// absolute encoder value at minimal joint positon
	g_minLinkEncoder :ARRAY[1..g_sArmNum, 1..g_sJntNum] OF DINT :=
		[5070618, 12248428, 9957376, 0, 0, 0, 0, 0,
		 4919708, 12165470, 13694272, 0, 0, 0, 0, 0,
		 9158200, 3936684, 16444112, 0, 0, 0, 0, 0,
		 13295020, 16357370, 9921792, 0, 0, 0, 0, 0];
		 
	// absolute encoder value at maximum joint positon
	g_maxLinkEncoder :ARRAY[1..g_sArmNum, 1..g_sJntNum] OF DINT :=
		[2939662, 5069530, 2375904, 0, 0, 0, 0, 0,
		2804134, 4974626, 6119888, 0, 0, 0, 0, 0,
		 6996994, 13526094, 8890176, 0, 0, 0, 0, 0,
		 11165812, 9145900, 2372960, 0, 0, 0, 0, 0];
	
	// absolute encoder value at calibrated positon
	g_caliLinkEncoder :ARRAY[1..g_sArmNum, 1..g_sJntNum] OF DINT :=
		[12427638, 8080000, 2375904, 15243664, 15283488, 7042832, 6950144, 7012272,
		12242476, 7980988, 6119888, 15217500, 15280288, 6866960, 6936528, 6826016,
		 16513242, 16579922, 8890176, 15265256, 15406944, 6400940, 6866960, 6902000,
		 3889656, 12177274, 2372960,15290800, 15066000, 6861290, 6710544, 6927488];
	
	 // if absolute encoder value cross zeros within joint motion range
	 // NOTICE: joint 7 is always 0.
	g_linkEncZeroCross :ARRAY[1..g_sArmNum, 1..g_sJntNum] OF INT :=
		[1, 0, 1, 1, 1, 1, 1, 1,
		 1, 0, 1, 1, 1, 1, 1, 1,
		 1, 1, 1, 1, 1, 1, 1, 1,
		 1, 0, 1, 1, 1, 1, 1, 1];
		 
	 // joint SDO address
	g_slaveArmNetID: ARRAY[1..4] OF T_AmsNetId:=['169.254.186.39.3.1','169.254.186.39.8.1','169.254.186.39.9.1','169.254.186.39.10.1'];
	g_slaveJointNetPort:ARRAY[1..g_sArmNum,1..g_sJntNum] OF UINT :=[
		1006,	1007,	1008,	2(1009),	3(1010),
		1006,	1007,	1008,	2(1009),	3(1010),
		1006,	1007,	1008,	2(1009),	3(1010),
		1006,	1007,	1008,	2(1009),	3(1010)];
		
//################ DO NOT modify parameters below ###########################
	// abolute encoder expanded limit buffer in case there is calibrtion error at limit position
	g_linkEncLimitBuffer : DINT := 100000;
	
	// absolute encoder direction
	g_asbEncoderDir :ARRAY[1..g_sJntNum] OF INT :=[1, -1, 1, 1, 1, 1, 1, 1];
	
	// flag if joint can rotate multiple cycles
	g_multipleCyclesJoint :ARRAY[1..g_sArmNum, 1..g_sJntNum] OF INT :=
		[0, 0, 0, 1, 1, 1, 1, 1,
		 0, 0, 0, 1, 1, 1, 1, 1,
		 0, 0, 0, 1, 1, 1, 1, 1,
		 0, 0, 0, 1, 1, 1, 1, 1];
		 
	// joint position at link encoder calibrated point
	g_linkEncCaliJntPos :ARRAY[1..g_sJntNum] OF LREAL :=
		[0.0, -PI/2 + 8*g_deg2rad, 0.581633, 5(0.0)];

	
END_VAR

// ---- GVLs/configs/robot6/GVL_CartJointEncoderCaliData_6.TcGVL
{attribute 'qualified_only'}
// Robot6 --joints parameters of setup arms
VAR_GLOBAL
	// absolute encoder value at minimal joint positon
	g_minLinkEncoder :ARRAY[1..g_cartJntNum] OF DINT :=[0, 0, 0, 0, 12912698, 863216, 13187303, 654894];
		 
	// absolute encoder value at maximum joint positon
	g_maxLinkEncoder :ARRAY[1..g_cartJntNum] OF DINT :=[0, 0, 0, 0, 10127418, 3841586, 15255509,16569304 ];
	
	// absolute encoder value at calibrated positon
	g_caliLinkEncoder :ARRAY[1..g_cartJntNum] OF DINT :=[0, 0, 0, 0, 12912698, 2352401, 15255509, 8612099];
	
	 // if absolute encoder value cross zeros within joint motion range
	g_linkEncZeroCross :ARRAY[1..g_cartJntNum] OF INT :=[0, 0, 0, 0, 0, 0, 0, 1];
		 

	// abolute encoder expanded limit buffer in case there is calibrtion error at limit position
	g_linkEncLimitBuffer : DINT := 100000;

	// absolute encoder direction
	g_asbEncoderDir :ARRAY[1..g_cartJntNum] OF INT :=[1, 1, 1, 1, -1, 1, -1, -1];
													
	// flag if joint can rotate multiple cycles
	g_multipleCyclesJoint :ARRAY[1..g_cartJntNum] OF INT :=[0, 0, 0, 0, 0, 0, 0, 0];
		 
	// joint position at link encoder calibrated point
	g_linkEncCaliJntPos :ARRAY[1..g_cartJntNum] OF LREAL :=[0.0, 0.0, 0.0, 0.0, 0.0, 0.0, 0, 0.0];
	
	 // joint SDO address
	g_slaveCartNetID: T_AmsNetId:='169.254.186.39.7.1';
	g_slaveCartJointNetPort:ARRAY[1..g_cartJntNum] OF UINT :=[1005,	1004,	1003,	1002,	1001,   1006,  1007,  1008];

END_VAR

// ---- GVLs/configs/robot6/GVL_SetupArmDynamics_6.TcGVL
{attribute 'global_init_slot' := '49992'}
{attribute 'qualified_only'}
// Robot6 --dynamic parameters of setup arms
VAR_GLOBAL 
	(* setup joint5 gravity parameters. last 5 parameters are defined in slave arm dynamic
	% graParam=[ 9.8*mx0,...
	%            4.92539*m1 + 4.92539*m2 + 4.92539*m3 + 7.8853*m4 + 7.8853*m5 + 9.70463*mx3 - 9.8*my0 - 1.3639*my3 + 9.8*mz1,...
	%            9.8*m5,...
	%            0.41601*m2 + 0.41601*m3 + 0.0000216012*m4 + 0.0000216012*m5 + 9.8*mx1 - 1.3639*mx3 - 9.70463*my3,...
	%            9.8*mz2 - 9.8*my5 - 9.8*my1 + 9.8*mz3 + 9.8*mz4,...
	%            2.19651*m3 + 2.19651*m4 + 0.00000258969*m5 + 8.64766*mx2 - 4.61063*my2 + 9.8*my4 + 9.8*mz5,...
	%            1.1711*m3 + 1.1711*m4 + 0.00000122416*m5 + 4.61063*mx2 - 9.8*mx4 - 9.8*mx5 + 8.64766*my2]';
	*)				
	//setup joint5 gravity parameters
	g_setupJnt5GravityParam :ARRAY[1..4,1..2] OF REAL := 
	[ 0.0000,   54.4806,
	  0.0196,   61.5623,
	  0.0196,   65.0026,
	  0.0196,   59.3080 ];

	(* setup joint3 gravity parameters
	 graParams = [p1,p2,p3,p4]
	 gravity = p1*q^3 + p2*q^2 + p3^q + p4
	 q(- [q0,q1]*)
 	// setup joint3 gravity parameter
	g_setupJnt3GravityParams :ARRAY[1..4, 1..4] OF LREAL :=
	[17452.1, -4008.76, 401.477, -117.096,
	 8476.95, -1240.58, 104.752, -105.76,
	 14956.5, -4297.99, 622.564, -131.776,
	 14926.3, -2807.93, 154.175, -103.6];
	 
	(* setup joint3 friction parameters
	 graParams = [p1mp2,p3,p4]
	 friciton = p1*q^3 + p2*q^2 + p3^q + p4
	 q(- [q0,q1]*)
 	// setup joint3 friction parameter
	g_setupJnt3FrictionParams :ARRAY[1..4, 1..4] OF LREAL :=
	[ -18790.6, 5987.36, -582.149, 60.6865,
	  -19818.6, 7327.61, -903.65, 81.3597,
	-60054.7, 22353.3, -2711.22, 147.637,
	-25150.3, 8097.23, -822.128, 75.4573];
	
	g_setupJnt3GravityPosRange :ARRAY[1..4, 1..2] OF REAL :=
	[0.0189, 	0.1789,
	 0.0182,    0.1784,
	 0.0189,    0.1789,
	 0.0189,    0.1789];
 	
	 
	// joint gravity offset
	g_setupJntGravityOffset :ARRAY[1..4,1..5] OF REAL := 
	[0, 0, 0, 0,  0,
	 0, 0, 0, 0,  0,
	 0, 0, 0, 0,  0,
	 0, 0, 0, 0,  0];

END_VAR

// ---- GVLs/configs/robot6/GVL_SetupJointEncoderCaliData_6.TcGVL
{attribute 'qualified_only'}
// Robot6 --joints parameters of setup arms
VAR_GLOBAL
	// absolute encoder value at minimal joint positon
	g_minLinkEncoder :ARRAY[1..g_sArmNum, 1..g_setupJntNum] OF DINT :=
		[15154005, 20642140, 2227846, 14466277, 9101921,
		 7319087, 17242128, 3319013, 14513407, 4923413,
		 1893735, 18952151, 5180416, 4939681, 4923413,
		 9631079, 15529480, 1114624, 6100507, 13177989];
		 
	// absolute encoder value at maximum joint positon
	g_maxLinkEncoder :ARRAY[1..g_sArmNum, 1..g_setupJntNum] OF DINT :=
		[3111223, 22098100, 3018537, 12898665, 1110933,
		 12036590, 18682052, 4122128, 12917951, 13714539,
		 6546979, 20395036, 14538137, 9477397, 13695977,
		 14360335, 16982188, 1934331, 4520019, 5314321];
	
	// absolute encoder value at calibrated positon
	g_caliLinkEncoder :ARRAY[1..g_sArmNum, 1..g_setupJntNum] OF DINT :=
		[746400, 20642329, 3019248, 5038400, 13414000,
		 9701120, 17236017, 4139006, 4959720, 9316700,
		 4250150, 18942693, 5244862, 9246550, 9290488,
		 11982000, 15555555, 1917113, 13457900, 991280];
	
	 // if absolute encoder value cross zeros within joint motion range
	g_linkEncZeroCross :ARRAY[1..g_sArmNum, 1..g_setupJntNum] OF INT :=
		[1, 0, 0, 0, 1,
		 0, 0, 0, 1, 0,
		 0, 0, 0, 0, 0,
		 0, 0, 0, 1, 1];
		 
//################ DO NOT modify parameters below ###########################
	// abolute encoder expanded limit buffer in case there is calibrtion error at limit position
	g_linkEncLimitBuffer : DINT := 100000;

	// absolute encoder direction
	g_asbEncoderDir :ARRAY[1..g_setupJntNum] OF INT :=[-1, -1, -1, 1, -1];
													
	// flag if joint can rotate multiple cycles
	g_multipleCyclesJoint :ARRAY[1..g_sArmNum, 1..g_setupJntNum] OF INT :=
		[0, 0, 0, 0, 0,
		 0, 0, 0, 0, 0,
		 0, 0, 0, 0, 0,
		 0, 0, 0, 0, 0];
		 
	// joint position at link encoder calibrated point
	g_linkEncCaliJntPos :ARRAY[1..g_sArmNum, 1..g_setupJntNum] OF LREAL :=
		[-140*g_deg2Rad, 0.779, 0.0, 90.0*g_deg2Rad, 0.0,
		 -115*g_deg2Rad, 0.607, 0.0, 90.0*g_deg2Rad, 0.0,
		 -65*g_deg2Rad, 0.607, 0.0, 90.0*g_deg2Rad, 0.0,
 		 -40*g_deg2Rad, 0.779, 0.0, 90.0*g_deg2Rad, 0.0];
	

END_VAR

// ---- GVLs/configs/robot6/GVL_SlaveArmDynamics_6.TcGVL
{attribute 'global_init_slot' := '49992'}
{attribute 'qualified_only'}
// Robot6 --dynamic parameters of slave arms
VAR_GLOBAL CONSTANT
	// arm gravity parameters
(*graParam=[ 9.8*m5,...
           0.41601*m2 + 0.41601*m3 + 0.0000216012*m4 + 0.0000216012*m5 + 9.8*mx1 - 1.3639*mx3 - 9.70463*my3,...
           9.8*mz2 - 9.8*my5 - 9.8*my1 + 9.8*mz3 + 9.8*mz4,...
           2.19651*m3 + 2.19651*m4 + 0.00000258969*m5 + 8.64766*mx2 - 4.61063*my2 + 9.8*my4 + 9.8*mz5,...
          1.1711*m3 + 1.1711*m4 + 0.00000122416*m5 + 4.61063*mx2 - 9.8*mx4 - 9.8*mx5 + 8.64766*my2]'
*)			
	// robot No.4
	g_gravityParam :ARRAY[1..4,1..5] OF REAL := 
	[ 7.5951,    1.6336,   -4.2417,    9.4106,    4.7289,
	  7.4741,    3.7472,   -4.4567,   10.5517,    7.6095,
	  7.6732,    3.7472,   -4.4458,    9.6721,    7.2742,
	  7.4582,    3.5688,   -3.7215,    9.2746,    5.7641];
	 
	g_gravityTrocar :ARRAY[1..5] OF REAL :=[0.1661, -0.4124,  0.0964,   -0.7987,   -0.6999 ];
	g_gravityInstrument :ARRAY[1..5] OF REAL :=[ 3.1217,  -0.3099,   0.0778,   -1.2498,   -0.8041];
	g_gravityEndoscope :ARRAY[1..5] OF REAL :=[10.8619,  -0.8575,   -1.0274,   -0.2425,   -0.0869];
	
	// joint friction(with instrument mounted)
	g_slaveJntFriction :ARRAY[1..g_sArmNum, 1..g_sJntNum] OF LREAL :=
			[ 5.3354,    9.5437,    4.6271,  0.03, 0.03, 0.03, 0.03, 0,
			  4.5927,    9.6040,    3.7367, 0.03, 0.03, 0.03, 0,
		      4.3557,    8.4286,    5.9078,  0.03, 0.03, 0.03, 0.03, 0,
              4.1447,    7.2202,    6.8253,  0.03, 0.03, 0.03, 0.03, 0	 ];
			  
	//################ DO NOT modify parameters below ###########################
	//################ dynamic reference model parameters below ###########################
	// link mass [m1, m2, m3, m4, m5]
	g_linkMass :ARRAY[1..5] OF LREAL :=[5.6565, 1.4613, 1.149, 1.5362, 0.6679] ;
	
	// lin center of amss
	g_linkCOM :ARRAY[1..5,1..3] OF LREAL :=  [ 0.0566,    0.0302,   -0.4685,
											   0.1191,   -0.0011,   -0.0588,
											   0.1238,    0.0003,   -0.0120,
											   0.0427,    0.0924,   -0.0004,
											   -0.0262,        0,   -0.0292];
	// link  inertial
    // [Ixx,Iyy,Izz, Ixy,Ixz, Iyz]
 	g_linkInertia :ARRAY[1..5,1..6] OF LREAL :=[0.0735,    0.0738,    0.0144,    0.0016,   -0.0000,   -0.0079,
												0.0016,    0.0190,    0.0185,         0,    0.0027,         0,
											   0.0009,    0.0167,    0.0166,         0,    0.0012,         0,
												0.0009,    0.0167,    0.0166,         0,    0.0012,         0,
											  0.0009,    0.0167,    0.0166,         0,    0.0012,         0];

	
	//  motor inertial at link size
	g_motorInertia :ARRAY[1..3] OF LREAL := [0.00004487, 0.00004487, 0.0000002280];
	
END_VAR

// ---- GVLs/configs/robot6/GVL_SlaveJointEncoderCaliData_6.TcGVL
{attribute 'qualified_only'}
// Robot6 --joints parameters of slave arms
VAR_GLOBAL CONSTANT
	// absolute encoder value at minimal joint positon
	g_minLinkEncoder :ARRAY[1..g_sArmNum, 1..g_sJntNum] OF DINT :=
		[9015451, 13207807, 650879, 0, 0, 0, 0, 0,
		 4890935, 9185623, 506623, 0, 0, 0, 0, 0,
		 712149, 4893469, 13158055, 0, 0, 0, 0, 0,
		 9022699, 13304191, 8138925, 0, 0, 0, 0, 0];
		 
	// absolute encoder value at maximum joint positon
	g_maxLinkEncoder :ARRAY[1..g_sArmNum, 1..g_sJntNum] OF DINT :=
		[6982407, 4260603, 9942895, 0, 0, 0, 0, 0,
		 2838445, 72017, 9799471, 0, 0, 0, 0, 0,
		 15438395, 12569941, 5587336, 0, 0, 0, 0, 0,
		 7017365, 4223351, 568399, 0, 0, 0, 0, 0];
	
	// absolute encoder value at calibrated positon
	g_caliLinkEncoder :ARRAY[1..g_sArmNum, 1..g_sJntNum] OF DINT :=
		[16348942, 6700, 9921200, 99713, 16623440, 8382220, 16654192, 8367312,
		 12305300, 12521700, 9764288, 16649696, 16555424, 8487936, 8451400, 8474272,
		 8116240, 8266990, 5574900, 16658032, 16560944, 8162864, 8354600, 2283056,
		 16416000, 16775600, 573808, 16553408, 16578880, 8005370, 8459520, 8439376];
	
	 // if absolute encoder value cross zeros within joint motion range
	 // NOTICE: joint 7 is always 0.
	g_linkEncZeroCross :ARRAY[1..g_sArmNum, 1..g_sJntNum] OF INT :=
		[1, 1, 0, 1, 1, 1, 1, 1,
		 1, 1, 0, 1, 1, 1, 1, 1,
		 0, 0, 1, 1, 1, 1, 1, 1,
		 1, 1, 1, 1, 1, 1, 1, 1];
		 
	 // joint SDO address
	g_slaveArmNetID: ARRAY[1..4] OF T_AmsNetId:=['169.254.186.39.3.1','169.254.186.39.8.1','169.254.186.39.9.1','169.254.186.39.10.1'];
	g_slaveJointNetPort:ARRAY[1..g_sArmNum,1..g_sJntNum] OF UINT :=[
		1006,	1007,	1008,	2(1009),	3(1010),
		1006,	1007,	1008,	2(1009),	3(1010),
		1006,	1007,	1008,	2(1009),	3(1010),
		1006,	1007,	1008,	2(1009),	3(1010)];
		
//################ DO NOT modify parameters below ###########################
	// abolute encoder expanded limit buffer in case there is calibrtion error at limit position
	g_linkEncLimitBuffer : DINT := 100000;
	
	// absolute encoder direction
	g_asbEncoderDir :ARRAY[1..g_sJntNum] OF INT :=[1, -1, 1, 1, 1, 1, 1, 1];
	
	// flag if joint can rotate multiple cycles
	g_multipleCyclesJoint :ARRAY[1..g_sArmNum, 1..g_sJntNum] OF INT :=
		[0, 0, 0, 1, 1, 1, 1, 1,
		 0, 0, 0, 1, 1, 1, 1, 1,
		 0, 0, 0, 1, 1, 1, 1, 1,
		 0, 0, 0, 1, 1, 1, 1, 1];
		 
	// joint position at link encoder calibrated point
	g_linkEncCaliJntPos :ARRAY[1..g_sJntNum] OF LREAL :=
		[0.0, -PI/2 + 8*g_deg2rad, 0.581633, 5(0.0)];

	
END_VAR

// ---- GVLs/GVL_interactUI.TcGVL
{attribute 'qualified_only'}
VAR_GLOBAL
	//read from UI
	//surgical status: true surgical start   false surgical finshed
	g_surgicalStatus : BOOL;

	//surgical site selection
	g_surgicalSite : UINT;

	//surgical location selection
	g_surgicalLocation : UINT;

	//stand column height limit : design 1805mm - 2495mm 
	g_heightLimit : UINT;
	g_heightLimitFromUI : UINT;
	g_heightLimitEnbale : BOOL;
	
	//ui control button enable
	g_uiCtrl : ST_uiControl;

	//ui send reset fault
	g_uiFaultReset : UINT;

	//write UI 
	//error code ID
	g_errIdType3 : UDINT;
	g_errIdType2 : UDINT;
	g_errIdType1 : UDINT;
	g_errIdType0 : UDINT;
	
	//instrument information
	g_instruInformatiom :ARRAY[1..4] OF  ST_instruInfomation;
	
	//UPS power supply mode : line voltage supply : 1 , battery powered : 2
	g_powerSupplyModeUPS : UINT;
	
	//UPS dump energy
	g_dumpEnergyUPS : UINT:=51;
	
	//ui shutdown button enable
	g_uiPowerOffEnable : BOOL;
	
	//plc confirm shutdown
	g_plcPowerOffEnable : BOOL:=FALSE;
	
	//joystick enable tip : true trigger
	g_joystickEnableTip : BOOL;
	
	//stop button signal : 0 press  , 1 No press
	g_stopButtonFormUI : UINT:=1;

	//PLC  version
	g_plcVersion : STRING := g_SWVersion;

	//Surgical guidance
	g_cartOperation : ST_cartOperation;
	
	//robot state  machine
	g_armStateMachine : ST_robotStateMachine;
	
	//scope gravity angle
	g_scopeGravityAngle : REAL;
	
	//scope type
	g_scopeType : INT;

	//fault tone current error type : 0 No fault , 1 low-level , 2 medium-level , 3 height-level
	g_curErrType : UINT;
	
	//30° endoscope face up or face down
	g_scopeUpDown : UINT := 1;
	
	//joystick signal  read RS232 data from UI
	g_joystickSignalArray : ARRAY[0..21] OF USINT;
	
	//joystick trigger
	g_joysticksTrigger : BOOL;
	
	//0: init status 1: checking 2:check succeed 3: check failed
	g_slaveSelfCheckStatus : UINT; 
	g_salveSelfCheckEnable : BOOL;
	
	//arm in disable status : 0 No disable , 1-4 number  corresponds to arms 1-4
	g_armIsDisable : UINT:=0;
	
	//the patient side has recover error flag
	g_slaveRecoverErrFlag : INT;

	//the patient side runs separately
	g_slaveRunAlone : BOOL;

	//trocar status : 0 No trocar , 1 have trocar
	g_trocarStatus : BOOL;

	//heartbeat signal
	g_heartBeat : INT;
	
	//left-right eye switch、0Left eye , 1 right eye
	g_switchLeftRightEye : INT;
	
	//the pop-up fault code is displayed
	g_popupErrorArm1 : ARRAY [0..2] OF UDINT;
	g_popupErrorArm2 : ARRAY [0..2] OF UDINT;
	g_popupErrorArm3 : ARRAY [0..2] OF UDINT;
	g_popupErrorArm4 : ARRAY [0..2] OF UDINT;
	g_popupRefresh : ARRAY [1..4] OF UINT;
	
	//instrument out of sight
	g_instruOutScope : ARRAY [1..4] OF BOOL;
	
	//arm is adjustment
	g_armIsAdjustment : ARRAY [1..4] OF UINT;
	
	//instrument max used record
	g_InstruSeriesRecord:ARRAY [1..100] OF ULINT;
END_VAR

// ---- GVLs/GVL_MathDefine.TcGVL
VAR_GLOBAL CONSTANT
	g_smallNum :LREAL := 1E-8;
	g_smallAng :LREAL := 0.0001*PI/180;
	g_largeNum: LREAL :=1E16;
	g_deg2Rad :LREAL := pi/180.0;
	g_rad2Deg :LREAL := 180.0/pi;
	g_2pi :LREAL :=2*PI;
	
	g_eye3d :Mat3d:=[1, 0, 0,
					 0, 1, 0,
					 0, 0, 1];
	g_eye4d :Mat4d:=[1, 0, 0, 0,
					 0, 1, 0, 0,
					 0, 0, 1, 0,
					 0, 0, 0, 1];
	g_zeroMat3d :Mat3d:=[9(0)];
	g_zeroMat35 :Mat35:=[15(0)];
	g_zeroMat6d :Mat6d:=[36(0)];
	g_zeroMat7d :Mat7d:=[49(0)];
	g_eye7d :Mat7d:=[1, 0, 0, 0, 0, 0, 0, 
					 0, 1, 0, 0, 0, 0, 0, 
					 0, 0, 1, 0, 0, 0, 0, 
					 0, 0, 0, 1, 0, 0, 0,
					 0, 0, 0, 0, 1, 0, 0,
					 0, 0, 0, 0, 0, 1, 0,
					 0, 0, 0, 0, 0, 0, 1];
	
	g_zeroVec2d :Vec2d:= [2(0)];
	
	g_zeroVec3i :Vec3i:= [3(0)];
	g_zeroVec3d :Vec3d:= [3(0)];
	g_onesVec3d: Vec3d:=[3(1)];
	
	g_zeroVec4b :Vec4b := [4(FALSE)];
	
	g_zeroVec6d: Vec6d:=[6(0)];
	g_onesVec6d: Vec6d:=[6(1)];
	g_zeroVec6b: Vec6b:=[6(FALSE)];
	g_onesVec6b: Vec6b:=[6(TRUE)];
	
	g_zeroVec5d: Vec5d:=[5(0)];
	g_onesVec5d: Vec5d:=[5(1.0)];
	g_zeroVec5i: Vec5i:=[5(0)];
	g_onesVec5i: Vec5i:=[5(1)];
	
	g_zeroVec7d: Vec7d:=[7(0)];
	g_onesVec7d: Vec7d:=[7(1.0)];
	g_zeroVec7i: Vec7i:=[7(0)];
	g_onesVec7i: Vec7i:=[7(1)];
	g_zeroVec8b: Vec8b:=[8(FALSE)];
	g_onesVec8b: Vec8b:=[8(TRUE)];
	g_zeroVec8d: Vec8d:=[8(0)];
	g_onesVec8d: Vec8d:=[8(1.0)];
	g_zeroVec8i: Vec8i:=[8(0)];
	g_onesVec8i: Vec8i:=[8(1)];
	g_initCurVec8d :Vec8d:=[8(250)];
	
	g_setupAllPosMode:Vec5i:=[5(DriverOPMode_Pos)];
	g_setupAllTrqMode:Vec5i:=[5(DriverOPMode_Trq)];
	g_slaveAllPosMode:Vec8i:=[8(DriverOPMode_Pos)];
	g_slaveAllTrqMode:Vec8i:=[8(DriverOPMode_Trq)];
	g_slaveAllPosTrqMode:Vec8i:=[8(DriverOPMode_PosTrq)];
	
	
END_VAR

// ---- GVLs/GVL_SafetyLogData.TcGVL
//{attribute 'qualified_only'}
VAR_GLOBAL CONSTANT
	g_maxNum:INT:=5;
	g_maxArmNum:INT:=4;
	g_maxArmJoint:INT:=13; g_maxCartJoint:INT:=8;
	g_cartNum:UDINT:=5;
	MAX_CSV_ROWS 			: UDINT := 10000;(*最大行数(任务周期为20ms)即10分钟的buffer*)
	MAX_CSV_COLUMNS 		: UDINT := 130;(*最大列数*)
	MAX_CSV_FIELD_LENGTH	: UDINT := 35;(*每个字段的字符长度*)
	MAX_CSV_RING_BUFFER		: UDINT := 5;
	g_JointNetPort:ARRAY[1..g_maxArmJoint] OF UINT :=[
		1002,    1002,	1003,	1004,	1005,	1006,	1007,	1008,	2(1009),	3(1010)];
END_VAR

VAR_GLOBAL
	g_arrayErrCodeArm:ARRAY [1..g_maxNum] OF ARRAY [0..100] OF UDINT;	
	g_zeroInstruRecord :ARRAY [1..100] OF ULINT;
END_VAR

// ---- GVLs/GVL_SafetyParameters.TcGVL
//{attribute 'qualified_only'}
{attribute 'global_init_slot' := '49991'}
VAR_GLOBAL CONSTANT
	// safety error counts threshold to trigger fault
	g_faultTriggerCounts :INT :=10;
	
	// arm joint safety error
	g_armMaxJntEncErr :vec13d:=[g_largeNum, g_largeNum, 0.010, 4(3*g_deg2Rad), 0.010, 5(10*g_deg2Rad)];
	g_armMaxJntFollowErr :vec13d:=[g_largeNum, g_largeNum, 0.010, 4(5*g_deg2Rad), 0.010, 5(170*g_deg2Rad)];
	
	//soft stiff control error---1028
	g_armMaxJntFollowErrSoftStiff :vec13d:=[g_largeNum, g_largeNum, 0.010, 2(5*g_deg2Rad),2(20*g_deg2Rad), 0.010, 5(170*g_deg2Rad)];
	
	//arm joint link encoder maximum and minimum values
	g_maxLinkEnc : vec13di:=[16777215, 2(67108863), 10(16777215)];
	g_minLinkEnc : vec13di:=[13(0)];
	
	//drive error word
	g_driveErrWord : UDINT:=32;
	
	// arm joint safety error
	g_safetyJntVel : vec13d:=[2(g_largeNum), 1.0, pi, pi, pi, pi, 0.6, 5(4*pi)];
	
	// joint limit buffer(outside of joint limit)
	g_armJntPosLimitBuffer :vec13d:=[10.0*g_deg2Rad,2(0.05),4(10.0*g_deg2Rad), 0.05, 5(0)];
	
	// joint position limit
	g_minJntPos: ARRAY[1..g_sArmNum,  1..13] OF LREAL:=[ (-140-50)*g_deg2Rad, 0.779-0.36,0.00,-1.2351,-1.6, -2.7,	-1.5-pi/2,	0.23, 5(-g_largeNum),
																	(-115-50)*g_deg2Rad, 0.607-0.36,0.00,-1.2351,-1.6, -2.7,	-1.5-pi/2,	0.23, 5(-g_largeNum),
																	(-65-50)*g_deg2Rad, 0.607-0.36,0.00,-1.2351,-1.6, -2.7,	-1.5-pi/2,	0.23, 5(-g_largeNum),
																	(-40-50)*g_deg2Rad, 0.779-0.36,0.00,-1.2351,-1.6, -2.7,	-1.5-pi/2,	0.23, 5(-g_largeNum)];	
	g_maxJntPos: ARRAY[1..g_sArmNum,  1..13] OF LREAL:=[ (-140+50)*g_deg2Rad, 0.779,0.200,4.5579,1.6, 2.7,	1.13-pi/2, 	0.58, 5(g_largeNum),
																	(-115+50)*g_deg2Rad, 0.607,0.200,4.5579,1.6, 2.7,	1.13-pi/2, 	0.58, 5(g_largeNum),
																	(-65+50)*g_deg2Rad, 0.607,0.200,4.5579,1.6, 2.7,	1.13-pi/2, 	0.58, 5(g_largeNum),
																	(-40+50)*g_deg2Rad, 0.779,0.200,4.5579,1.6, 2.7,	1.13-pi/2, 	0.58, 5(g_largeNum)];	
	
	//arm joint max current
	g_maxJntCurrent : vec13d:=[2(g_largeNum),8400,7600,8400,      8400,8400,      1500,300,300,300,300, 300];
	
	// rcp position deviation for safety check
	g_rcpDeviationThres :LREAL := 0.005;
	
	//max joint commend  saltation
	g_maxJntCmdSalta : vec13d:=[2(g_largeNum), 0.010, 5(5*g_deg2Rad), 5(35*g_deg2Rad)];
	
	//max joint encoder current  saltation
	g_maxJntCurSalta : vec13d:=[2(g_largeNum), 11(60000)];
	
	// setup joint limit buffer(outside of joint limit)
	g_setupJntPosLimitBuffer :Vec5d := [5.0*g_deg2Rad, 0.01, 0.01,  2(5.0*g_deg2Rad)];
	
	// slave arm cartesion control safety error 
	g_maxCartPoseErr :ARRAY [1..6] OF LREAL:=[0.010,0.010,0.010,90*g_deg2Rad,90*g_deg2Rad,90*g_deg2Rad];
	
	//instrument open angle maximum and minimum values
	g_maxInstruOpen:LREAL;
	g_minInstruOpen:LREAL;
	
	g_motPhieErrLimit:DINT:=20000;
	
	//motor deviation between command current and feedback current limit
	g_jntCurrentCtrlLimit : vec13d:=[2(g_largeNum), 1680, 1140, 3(1680), 200, 5(g_largeNum)];
	
	// cart joint safety check limit
	g_cartMaxJntEncErr :Vec8d:=[0.01,0.01,3*g_deg2Rad,3*g_deg2Rad,0.01,3*g_deg2Rad,0.01,3*g_deg2Rad];
	g_cartMaxJntFollowErr :Vec8d:=[0.01,0.01,3*g_deg2Rad,3*g_deg2Rad,0.01,3*g_deg2Rad,0.01,3*g_deg2Rad];
	g_cartMaxLinkEnc :Vec8di:=[4(1), 67108863,16777215,67108863,16777215] ;
	g_cartMinLinkEnc :Vec8di:=[4(1),  4(0)];
	g_cartMaxJntVel :Vec8d:=[0.0025*2,0.0025*2,2.3*2,2.3*2, 0.032, 10*g_deg2Rad, 0.10, 10*g_deg2Rad];
	g_cartMaxJntCurrent :Vec8d:=[1080*2,1080*2,19800*2,19800*2, 10000*2,3800*2,3800*2,3800*2];
	g_cartMinJntPos :Vec8d:=[0,		0,		1, 1,  0-0.01,		-35*g_deg2Rad,	0-0.02,		-165*g_deg2Rad];
	g_cartMaxJntPos :Vec8d:=[0.053,0.053,1, 1,  0.68+0.01, 35*g_deg2Rad,	0.5+0.02,	165*g_deg2Rad];
END_VAR

// ---- GVLs/GVL_SystemParameters.TcGVL
VAR_GLOBAL CONSTANT
		
	g_SWVersion : STRING := '2(1.0.0.1)';
	
	g_mArmNum :INT := 2;	
	g_mJntNum :INT := 7;	
	g_sArmNum :INT := 4;	
	g_sJntNum :INT := 8;
	g_setupJntNum :INT :=5;
	g_cartDofs :INT :=6;
	g_cartJntNum:INT :=8;
	
	
	
	// control loop interval for each task
	g_slaveArmCtrlCycleTime :LREAL :=0.00025;
	g_slaveArmCtrlFreq :LREAL :=1.0/g_slaveArmCtrlCycleTime;
	g_armDynamicCycleTime :LREAL := 0.001;
	g_armDynamicFreq :LREAL := 1.0/g_armDynamicCycleTime;
	g_setupArmCtrlCycleTime :LREAL := 0.001;
	g_setupArmCtrlFreq :LREAL := 1.0/g_setupArmCtrlCycleTime;
	g_cartCtrlCycleTime :LREAL := 0.001;
	g_cartCtrlFreq :LREAL := 1.0/g_cartCtrlCycleTime;
	
	// wait time before robot init  for ethercat to stablize 
	g_robotInitWaitTime : LREAL := 1.0;

	g_robotSafetyCheckWaitTime : LREAL :=3.0;
END_VAR

// ---- GVLs/Instrument/GVL_InstruCtrlParams.TcGVL
// NOTICE： Use m_instruTypeIdx in FB_Instrument as the array index to get data below
{attribute 'global_init_slot' := '49991'}
VAR_GLOBAL CONSTANT
	// master gripper angle limit
	g_maxMasterGripAngle :LREAL := 30*g_deg2Rad;
	g_minMasterGripAngle : LREAL :=0.0;
	g_masterGripForceStartAng :LREAL :=5*g_deg2Rad;
	
	// gripper angle corresponding to g_masterGripForceStartAng
	// make sure fingers are fully closed and have a initial force
	g_minSlaveGripAngle :LREAL := -20 * g_deg2Rad; 
	
	//ultrasound knife kinematics parameter
	g_uknifeGripTravel :LREAL:= 0.00353;
	g_uknifeGripDividAngle : LREAL := 17 * g_deg2Rad;
	g_uknifeMotorLead : LREAL := 0.025;
	g_uknifeLeverRatio : LREAL := 13.0/18.5;
	
	// prograsp kinematic parameters
	g_proGraspAB :LREAL :=2.8;
	g_proGraspBC :LREAL :=5.26;
	g_proGraspInitA :LREAL :=16.6*g_deg2Rad;;
	g_proGraspInitC :LREAL :=8.75*g_deg2Rad;
	
	g_proGrasp2AB :LREAL :=2.7;
	g_proGrasp2BC :LREAL :=5.245;
	g_proGrasp2InitA :LREAL :=16.13*g_deg2Rad;;
	g_proGrasp2InitC :LREAL :=8.21*g_deg2Rad;
	
	// instrument grip yaw compensation
	g_instruBacklashDir: ARRAY[1..5] OF INT :=[-1, -1, -1, 0, 0];
	g_instruGripYawCompAng :ARRAY[1..4] OF LREAL := [ 2*g_deg2rad,  4*g_deg2rad,  6*g_deg2rad,  8*g_deg2rad];
	g_instruGripYawCompForceLevel  :ARRAY[1..4] OF INT := [ 20, 40, 70, 101];
	
END_VAR

// ---- GVLs/Instrument/GVL_InstruTypeDefine.TcGVL
// NOTICE：this file would be defined as config file later
{attribute 'global_init_slot' := '49991'}
VAR_GLOBAL CONSTANT
	InstruTypeInfo_CadiereForceps :ST_InstruTypeInfo :=
	(m_InstruID:=7, m_isSingleFinger:=FALSE, m_energyType:=0, m_instruName:='Cadiere Forceps', m_instruNameCH:="无创抓钳", m_maxUseNum:=20,
	 m_rodLength:=0.5438, m_headLength:=0.0089, m_fingerLength:=0.0195, m_maxGripAngle:=45*g_deg2Rad,
	 m_k1:= 0.859649123, m_k2:=0.947368421, m_k3:=0.775510204,
	 m_rollLimit:=5.5, m_pitchLimit:=75*g_deg2Rad, m_yawLimit:=PI/2, m_normGripTrq := 150,
	 m_instruYawBacklash:=4*g_deg2Rad, m_instruPitchBachlash:=3*g_deg2Rad);
	 
	InstruTypeInfo_NeedleDriver :ST_InstruTypeInfo :=
	(m_InstruID:=8, m_isSingleFinger:=FALSE, m_energyType:=0, m_instruName:='Large Needle Driver', m_instruNameCH:="持针钳", m_maxUseNum:=20,
	 m_rodLength:=0.5438, m_headLength:=0.0089, m_fingerLength:=0.0096, m_maxGripAngle:=40*g_deg2Rad,
	 m_k1:= 0.824561404, m_k2:=0.947368421, m_k3:=0.808510638,
	 m_rollLimit:=5.5, m_pitchLimit:=75*g_deg2Rad, m_yawLimit:=PI/2, m_normGripTrq := 150,
	 m_instruYawBacklash:=4*g_deg2Rad, m_instruPitchBachlash:=3*g_deg2Rad);
	 
	InstruTypeInfo_MegaSCNeedleDriver :ST_InstruTypeInfo :=
	(m_InstruID:=9, m_isSingleFinger:=FALSE, m_energyType:=0, m_instruName:='Mega SutureCut Needle Driver', m_instruNameCH:="大号带剪刀持针钳", m_maxUseNum:=20,
	 m_rodLength:=0.5438, m_headLength:=0.01, m_fingerLength:=0.0109, m_maxGripAngle:=40*g_deg2Rad,
	 m_k1:= 1.070175439, m_k2:=0.947368421, m_k3:=0.590163934,
	 m_rollLimit:=5.5, m_pitchLimit:=75*g_deg2Rad, m_yawLimit:=PI/2, m_normGripTrq := 150,
	 m_instruYawBacklash:=4*g_deg2Rad, m_instruPitchBachlash:=3*g_deg2Rad);
	 
	 InstruTypeInfo_SCNeedleDriver :ST_InstruTypeInfo :=
	(m_InstruID:=10, m_isSingleFinger:=FALSE, m_energyType:=0, m_instruName:='Large SutureCut Needle Driver', m_instruNameCH:="带剪刀持针钳", m_maxUseNum:=20,
	 m_rodLength:=0.5438, m_headLength:=0.01, m_fingerLength:=0.011, m_maxGripAngle:=40*g_deg2Rad,
	 m_k1:= 1.070175439, m_k2:=0.947368421, m_k3:=0.590163934,
	 m_rollLimit:=5.5, m_pitchLimit:=75*g_deg2Rad, m_yawLimit:=PI/2, m_normGripTrq := 150,
	 m_instruYawBacklash:=4*g_deg2Rad, m_instruPitchBachlash:=3*g_deg2Rad);
	 
	 InstruTypeInfo_RoundTipScissors :ST_InstruTypeInfo :=
	(m_InstruID:=11, m_isSingleFinger:=FALSE, m_energyType:=0, m_instruName:='RoundTip Scissors', m_instruNameCH:="圆头直剪", m_maxUseNum:=20,
	 m_rodLength:=0.5438, m_headLength:=0.0089, m_fingerLength:=0.01102, m_maxGripAngle:=40*g_deg2Rad,
	 m_k1:= 0.842105263, m_k2:=0.947368421, m_k3:=0.791666667,
	 m_rollLimit:=5.5, m_pitchLimit:=75*g_deg2Rad, m_yawLimit:=PI/2, m_normGripTrq := 150, 
	 m_instruYawBacklash:=4*g_deg2Rad, m_instruPitchBachlash:=3*g_deg2Rad);
	 
	 InstruTypeInfo_ProGraspForceps :ST_InstruTypeInfo :=
	(m_InstruID:=12, m_isSingleFinger:=FALSE, m_energyType:=0, m_instruName:='Prograsp', m_instruNameCH:="细齿无创抓钳", m_maxUseNum:=20,
	 m_rodLength:=0.5438, m_headLength:=0.01065, m_fingerLength:=0.02773, m_maxGripAngle:=44.5*g_deg2rad,
	 m_k1:= 1.342105263, m_k2:=0.947368421, m_k3:=0.496732026,
	 m_rollLimit:=5.5, m_pitchLimit:=75*g_deg2Rad, m_yawLimit:=PI/2, m_normGripTrq := 150,
	 m_instruYawBacklash:=4*g_deg2Rad, m_instruPitchBachlash:=3*g_deg2Rad);
	 
	 InstruTypeInfo_MarylandForceps :ST_InstruTypeInfo :=
	(m_InstruID:=13, m_isSingleFinger:=FALSE, m_energyType:=2, m_instruName:='Maryland Bipolar Forceps', m_instruNameCH:="双极弧形电凝钳", m_maxUseNum:=20,
	 m_rodLength:=0.5438, m_headLength:=0.01065, m_fingerLength:=0.0195, m_maxGripAngle:=55*g_deg2Rad,
	 m_k1:= 1.070175439, m_k2:=0.947368421, m_k3:=0.590163934,
	 m_rollLimit:=5.5, m_pitchLimit:=75*g_deg2Rad, m_yawLimit:=PI/2, m_normGripTrq := 150,
	 m_instruYawBacklash:=4*g_deg2Rad, m_instruPitchBachlash:=3*g_deg2Rad);
	 
	 InstruTypeInfo_FenestratedForceps :ST_InstruTypeInfo :=
	(m_InstruID:=14, m_isSingleFinger:=FALSE, m_energyType:=2, m_instruName:='Fenestrated Bipolar Forceps', m_instruNameCH:="双极鸭嘴电凝钳", m_maxUseNum:=20,
	 m_rodLength:=0.5438, m_headLength:=0.01065, m_fingerLength:=0.0207, m_maxGripAngle:=55*g_deg2Rad,
	 m_k1:= 1.070175439, m_k2:=0.947368421, m_k3:=0.590163934,
	 m_rollLimit:=5.5, m_pitchLimit:=75*g_deg2Rad, m_yawLimit:=PI/2, m_normGripTrq := 150, 
	 m_instruYawBacklash:=4*g_deg2Rad, m_instruPitchBachlash:=3*g_deg2Rad);
	 
	 InstruTypeInfo_CurvedScissors :ST_InstruTypeInfo :=
	(m_InstruID:=15, m_isSingleFinger:=FALSE, m_energyType:=1, m_instruName:='Monopolar Curved Scissors', m_instruNameCH:="单极弧剪", m_maxUseNum:=20,
	 m_rodLength:=0.5438, m_headLength:=0.0091, m_fingerLength:=0.0130, m_maxGripAngle:=PI/3,
	 m_k1:= 0.842105263, m_k2:=0.947368421, m_k3:=0.75,
	 m_rollLimit:=5.5, m_pitchLimit:=75*g_deg2Rad, m_yawLimit:=PI/2, m_normGripTrq := 150,
	 m_instruYawBacklash:=4*g_deg2Rad, m_instruPitchBachlash:=3*g_deg2Rad);
	 
	 InstruTypeInfo_CauteryHook :ST_InstruTypeInfo :=
	(m_InstruID:=16, m_isSingleFinger:=TRUE, m_energyType:=1, m_instruName:='Permanent Cautery Hook', m_instruNameCH:="单极电钩", m_maxUseNum:=20,
	 m_rodLength:=0.5432, m_headLength:=0.00935, m_fingerLength:=0.01668, m_maxGripAngle:=0,
	 m_k1:= 0.964912281, m_k2:= 0.877192982, m_k3:=-0.663636364,
	 m_rollLimit:=5.5, m_pitchLimit:=75*g_deg2Rad, m_yawLimit:=PI/2, m_normGripTrq := 0,
	 m_instruYawBacklash:=8*g_deg2Rad, m_instruPitchBachlash:=3*g_deg2Rad);
	 
	 InstruTypeInfo_CauterySpatula :ST_InstruTypeInfo :=
	(m_InstruID:=17, m_isSingleFinger:=TRUE, m_energyType:=1, m_instruName:='Permanent Cautery Spatula', m_instruNameCH:="单极电铲", m_maxUseNum:=20,
	 m_rodLength:=0.5432, m_headLength:=0.00935, m_fingerLength:=0.01905, m_maxGripAngle:=0,
	 m_k1:= 0.964912281, m_k2:= 0.877192982, m_k3:=-0.663636364,
	 m_rollLimit:=5.5, m_pitchLimit:=75*g_deg2Rad, m_yawLimit:=PI/2, m_normGripTrq := 0,
	 m_instruYawBacklash:=8*g_deg2Rad, m_instruPitchBachlash:=3*g_deg2Rad);
	 
	 InstruTypeInfo_Endoscope :ST_InstruTypeInfo :=
	(m_InstruID:=20, m_isSingleFinger:=FALSE, m_energyType:=0, m_instruName:='Camera', m_instruNameCH:="内窥镜", m_maxUseNum:=100,
	 m_rodLength:=0.49, m_headLength:=0, m_fingerLength:=0, m_maxGripAngle:=0,
	 m_k1:= 1, m_k2:= 1, m_k3:=1,
	 m_rollLimit:=5.5, m_pitchLimit:=1*g_deg2Rad, m_yawLimit:=1*g_deg2Rad, m_normGripTrq := 0,
	 m_instruYawBacklash:=0, m_instruPitchBachlash:=0);
	 
	 
	 InstruTypeInfo_NewEndoscope :ST_InstruTypeInfo :=
	(m_InstruID:=31, m_isSingleFinger:=FALSE, m_energyType:=0, m_instruName:='Camera', m_instruNameCH:="内窥镜", m_maxUseNum:=100,
	 m_rodLength:=0.49, m_headLength:=0, m_fingerLength:=0, m_maxGripAngle:=0,
	 m_k1:= 1, m_k2:= 1, m_k3:=1,
	 m_rollLimit:=5.5, m_pitchLimit:=1*g_deg2Rad, m_yawLimit:=1*g_deg2Rad,
	 m_instruYawBacklash:=0, m_instruPitchBachlash:=0);
	 
	 InstruTypeInfo_UltrasoundKnifeS :ST_InstruTypeInfo :=
	(m_InstruID:=42, m_isSingleFinger:=FALSE, m_energyType:=3, m_instruName:='Ultrasonic Scalpel 45cm', m_instruNameCH:="超声刀 46cm", m_maxUseNum:=1,
	 m_rodLength:=0.46463, m_headLength:=0, m_fingerLength:=0, m_maxGripAngle:=PI/4,
	 m_k1:= 1, m_k2:= 1, m_k3:=1,
	 m_rollLimit:=g_largeNum, m_pitchLimit:=1*g_deg2Rad, m_yawLimit:=1*g_deg2Rad, m_normGripTrq := 150,
	 m_instruYawBacklash:=4*g_deg2Rad, m_instruPitchBachlash:=0);
	 
	 InstruTypeInfo_UltrasoundKnifeU :ST_InstruTypeInfo :=
	(m_InstruID:=43, m_isSingleFinger:=FALSE, m_energyType:=3, m_instruName:='Ultrasonic Scalpel 55cm', m_instruNameCH:="超声刀 55cm", m_maxUseNum:=1,
	 m_rodLength:=0.55225, m_headLength:=0, m_fingerLength:=0, m_maxGripAngle:=PI/4,
	 m_k1:= 1, m_k2:= 1, m_k3:=1,
	 m_rollLimit:=g_largeNum, m_pitchLimit:=1*g_deg2Rad, m_yawLimit:=1*g_deg2Rad, m_normGripTrq := 150,
	 m_instruYawBacklash:=4*g_deg2Rad, m_instruPitchBachlash:=0);
	 
	 InstruTypeInfo_TipUpFenestratedGrasper :ST_InstruTypeInfo :=
	(m_InstruID:=44, m_isSingleFinger:=FALSE, m_energyType:=0, m_instruName:='Tip-Up Fenestrated Grasper', m_instruNameCH:="鸭嘴抓钳", m_maxUseNum:=20,
	 m_rodLength:=0.5438, m_headLength:=0.01065, m_fingerLength:=0.032, m_maxGripAngle:=PI/3,
	 m_k1:= 1.29824561403509, m_k2:=0.947368421052632, m_k3:=0.513513513513513,
	 m_rollLimit:=5.5, m_pitchLimit:=75*g_deg2Rad, m_yawLimit:=PI/2, m_normGripTrq := 150,
	 m_instruYawBacklash:=4*g_deg2Rad, m_instruPitchBachlash:=3*g_deg2Rad);
	 
	 InstruTypeInfo_MegaNeedleDriver :ST_InstruTypeInfo :=
	(m_InstruID:=45, m_isSingleFinger:=FALSE, m_energyType:=0, m_instruName:='Mega Needle Driver', m_instruNameCH:="大号持针钳", m_maxUseNum:=20,
	 m_rodLength:=0.5438, m_headLength:=0.011, m_fingerLength:=0.0130, m_maxGripAngle:=PI/6,
	 m_k1:=1.28070175438596 , m_k2:=0.929824561403509, m_k3:=0.520547945205479,
	 m_rollLimit:=5.5, m_pitchLimit:=75*g_deg2Rad, m_yawLimit:=PI/2, m_normGripTrq := 150,
	 m_instruYawBacklash:=4*g_deg2Rad, m_instruPitchBachlash:=3*g_deg2Rad);
	 
	 InstruTypeInfo_DeBakeyForceps :ST_InstruTypeInfo :=
	(m_InstruID:=46, m_isSingleFinger:=FALSE, m_energyType:=0, m_instruName:='DeBakey Forceps', m_instruNameCH:="微型抓钳", m_maxUseNum:=20,
	 m_rodLength:=0.5438, m_headLength:=0.0089, m_fingerLength:=0.0120, m_maxGripAngle:=PI/6,
	 m_k1:= 0.824561403508772, m_k2:=0.947368421052632, m_k3:=0.808510638297872,
	 m_rollLimit:=5.5, m_pitchLimit:=75*g_deg2Rad, m_yawLimit:=PI/2, m_normGripTrq := 150,
	 m_instruYawBacklash:=4*g_deg2Rad, m_instruPitchBachlash:=3*g_deg2Rad);
	 
	 InstruTypeInfo_BlackDiamondForceps :ST_InstruTypeInfo :=
	(m_InstruID:=47, m_isSingleFinger:=FALSE, m_energyType:=0, m_instruName:='Black Diamond Micro Forceps', m_instruNameCH:="黑钻微型钳", m_maxUseNum:=20,
	 m_rodLength:=0.5438, m_headLength:=0.0089, m_fingerLength:=0.010, m_maxGripAngle:=PI/6,
	 m_k1:= 0.8245614035087, m_k2:=0.947368421052632, m_k3:=0.808510638297872,
	 m_rollLimit:=5.5, m_pitchLimit:=75*g_deg2Rad, m_yawLimit:=PI/2, m_normGripTrq := 150,
	 m_instruYawBacklash:=4*g_deg2Rad, m_instruPitchBachlash:=3*g_deg2Rad);
	 
	 InstruTypeInfo_PottsScissors :ST_InstruTypeInfo :=
	(m_InstruID:=48, m_isSingleFinger:=FALSE, m_energyType:=0, m_instruName:='Potts Scissors', m_instruNameCH:="波茨手术剪", m_maxUseNum:=20,
	 m_rodLength:=0.5438, m_headLength:=0.0089, m_fingerLength:=0.0110, m_maxGripAngle:=22*g_deg2Rad,
	 m_k1:= 0.824561403508772, m_k2:=0.947368421052632, m_k3:=0.808510638297872,
	 m_rollLimit:=5.5, m_pitchLimit:=75*g_deg2Rad, m_yawLimit:=PI/2, m_normGripTrq := 150,
	 m_instruYawBacklash:=4*g_deg2Rad, m_instruPitchBachlash:=3*g_deg2Rad);
	 
	 InstruTypeInfo_CurvedBipolarDissector :ST_InstruTypeInfo :=
	(m_InstruID:=49, m_isSingleFinger:=FALSE, m_energyType:=2, m_instruName:='Curved Bipolar Dissector', m_instruNameCH:="双极分离电凝钳", m_maxUseNum:=20,
	 m_rodLength:=0.5438, m_headLength:=0.01065, m_fingerLength:=0.022, m_maxGripAngle:=PI/4,
	 m_k1:= 1.07017543859649, m_k2:=0.947368421052632, m_k3:=0.59016393442623,
	 m_rollLimit:=5.5, m_pitchLimit:=75*g_deg2Rad, m_yawLimit:=PI/2, m_normGripTrq := 150,
	 m_instruYawBacklash:=4*g_deg2Rad, m_instruPitchBachlash:=3*g_deg2Rad);
	 
	 InstruTypeInfo_MicroBipolarForceps :ST_InstruTypeInfo :=
	(m_InstruID:=50, m_isSingleFinger:=FALSE, m_energyType:=2, m_instruName:='Micro Bipolar Forceps', m_instruNameCH:="双极微型镊", m_maxUseNum:=20,
	 m_rodLength:=0.5438, m_headLength:=0.01065, m_fingerLength:=0.014, m_maxGripAngle:=PI/4,
	 m_k1:= 1.07017543859649, m_k2:=0.947368421052632, m_k3:=0.59016393442623,
	 m_rollLimit:=5.5, m_pitchLimit:=75*g_deg2Rad, m_yawLimit:=PI/2, m_normGripTrq := 150,
	 m_instruYawBacklash:=4*g_deg2Rad, m_instruPitchBachlash:=3*g_deg2Rad);
	 
	 InstruTypeInfo_ForceBipolar :ST_InstruTypeInfo :=
	(m_InstruID:=51, m_isSingleFinger:=FALSE, m_energyType:=0, m_instruName:='Force Bipolar', m_instruNameCH:="强力双极电凝钳", m_maxUseNum:=20,
	 m_rodLength:=0.5438, m_headLength:=0.01065, m_fingerLength:=0.024, m_maxGripAngle:=42*g_deg2Rad,
	 m_k1:= 1.28947368421053, m_k2:=0.947368421052632, m_k3:=0.517006802721088,
	 m_rollLimit:=5.5, m_pitchLimit:=75*g_deg2Rad, m_yawLimit:=PI/2, m_normGripTrq := 80, 
	 m_instruYawBacklash:=4*g_deg2Rad, m_instruPitchBachlash:=3*g_deg2Rad);
	 
	 InstruTypeInfo_MicroCauteryHook :ST_InstruTypeInfo :=
	(m_InstruID:=52, m_isSingleFinger:=FALSE, m_energyType:=0, m_instruName:='Micro Permanent Cautery Hook', m_instruNameCH:="小号单极电钩", m_maxUseNum:=20,
	 m_rodLength:=0.5432, m_headLength:=0.00935, m_fingerLength:=0.01668, m_maxGripAngle:=0,
	 m_k1:= 0.964912281, m_k2:= 0.877192982, m_k3:=-0.663636364,
	 m_rollLimit:=5.5, m_pitchLimit:=75*g_deg2Rad, m_yawLimit:=PI/2, m_normGripTrq := 0,
	 m_instruYawBacklash:=8*g_deg2Rad, m_instruPitchBachlash:=3*g_deg2Rad);
	 
	 g_instruTypeNum :INT :=24;
	 g_instruTypePool :ARRAY[1..g_instruTypeNum] OF ST_InstruTypeInfo :=
	 [InstruTypeInfo_CadiereForceps, 	InstruTypeInfo_NeedleDriver,  		InstruTypeInfo_MegaSCNeedleDriver, 	InstruTypeInfo_SCNeedleDriver,
	  InstruTypeInfo_RoundTipScissors,	InstruTypeInfo_ProGraspForceps,		InstruTypeInfo_MarylandForceps,		InstruTypeInfo_FenestratedForceps,
	  InstruTypeInfo_CurvedScissors,	InstruTypeInfo_CauteryHook,	 		InstruTypeInfo_CauterySpatula, 		InstruTypeInfo_Endoscope, InstruTypeInfo_NewEndoscope,
	  InstruTypeInfo_UltrasoundKnifeU, 	InstruTypeInfo_UltrasoundKnifeS,	InstruTypeInfo_TipUpFenestratedGrasper, 		InstruTypeInfo_MegaNeedleDriver, 
	  InstruTypeInfo_DeBakeyForceps, 	InstruTypeInfo_BlackDiamondForceps, 	InstruTypeInfo_PottsScissors, 	InstruTypeInfo_CurvedBipolarDissector,
	  InstruTypeInfo_MicroBipolarForceps,InstruTypeInfo_ForceBipolar, InstruTypeInfo_MicroCauteryHook];

	 
END_VAR

// ---- GVLs/SetupArms/GVL_SetupArmDynamics.TcGVL
{attribute 'global_init_slot' := '49992'}
{attribute 'qualified_only'}
// Robot3 --dynamic parameters of setup arms
VAR_GLOBAL 
	(* setup joint5 gravity parameters. last 5 parameters are defined in slave arm dynamic
	% graParam=[ 9.8*mx0,...
	%            4.92539*m1 + 4.92539*m2 + 4.92539*m3 + 7.8853*m4 + 7.8853*m5 + 9.70463*mx3 - 9.8*my0 - 1.3639*my3 + 9.8*mz1,...
	%            9.8*m5,...
	%            0.41601*m2 + 0.41601*m3 + 0.0000216012*m4 + 0.0000216012*m5 + 9.8*mx1 - 1.3639*mx3 - 9.70463*my3,...
	%            9.8*mz2 - 9.8*my5 - 9.8*my1 + 9.8*mz3 + 9.8*mz4,...
	%            2.19651*m3 + 2.19651*m4 + 0.00000258969*m5 + 8.64766*mx2 - 4.61063*my2 + 9.8*my4 + 9.8*mz5,...
	%            1.1711*m3 + 1.1711*m4 + 0.00000122416*m5 + 4.61063*mx2 - 9.8*mx4 - 9.8*mx5 + 8.64766*my2]';
	*)				
	//setup joint5 gravity parameters
	g_setupJnt5GravityParam :ARRAY[1..4,1..2] OF REAL := 
	[ 0.0000,   54.4806,
	  0.0196,   61.5623,
	  0.0196,   65.0026,
	  0.0196,   59.3080 ];

	(* setup joint3 gravity parameters
	 graParams = [p1mp2,p3,p4]
	 gravity = p1*q^3 + p2*q^2 + p3^q + p4
	 q(- [q0,q1]*)
 	// setup joint3 gravity parameter
	g_setupJnt3GravityParams :ARRAY[1..4, 1..4] OF LREAL :=
	[13129.9, -3010.8, 300.188, -99.7871,
	 14085.9, -3787.37, 476.955, -104.313,
	  6440.78, -1524.39, 415.869, -117.102,
	 22097.9, -5714.59, 558.077, -104.732];
	 
	(* setup joint3 friction parameters
	 graParams = [p1mp2,p3,p4]
	 friciton = p1*q^3 + p2*q^2 + p3^q + p4
	 q(- [q0,q1]*)
 	// setup joint3 friction parameter
	g_setupJnt3FrictionParams :ARRAY[1..4, 1..4] OF LREAL :=
	[-11173.7, 3888.25, -491.555, 79.4495,
	 -17709.9, 6947.19, -897.825, 94.243,
	 -49343.5, 18899.5, -2449.52, 166.011,
	-11537.6, 3698.16, -380.906, 51.8712];
	
	g_setupJnt3GravityPosRange :ARRAY[1..4, 1..2] OF REAL :=
	[0.0189, 	0.1789,
	 0.0182,    0.1784,
	 0.0189,    0.1789,
	 0.0189,    0.1789];
 	
	// joint gravity offset
	g_setupJntGravityOffset :ARRAY[1..4,1..5] OF REAL := 
	[0, 0, 0, 0,  0,
	 0, 0, 0, 0,  0,
	 0, 0, 0, 0,  0,
	 0, 0, 0, 0,  0];

END_VAR

// ---- GVLs/SetupArms/GVL_SetupJointEncoderCaliData.TcGVL
{attribute 'qualified_only'}
// Robot3 --joints parameters of setup arms
VAR_GLOBAL
	// absolute encoder value at minimal joint positon
	g_minLinkEncoder :ARRAY[1..g_sArmNum, 1..g_setupJntNum] OF DINT :=
		[5813168, 22663264, 1978132, 1938100, 13659124,
		 13487924, 17543781, 3084321, 10238892, 1028618,
		  3186404, 15837168, 878439, 6065586, 9487992,
		  553720, 24385008, 4169014, 6084058, 984346];
		 
	// absolute encoder value at maximum joint positon
	g_maxLinkEncoder :ARRAY[1..g_sArmNum, 1..g_setupJntNum] OF DINT :=
		[1055544, 21209065, 1176866, 385208, 4921448,
		 8781908, 16093586, 2285859, 8654922, 9089506,
		 15289572, 14389054, 85603, 4478314, 767644,
		  12599264, 22936561, 3373290, 4489778, 9055426];
	
	// absolute encoder value at calibrated positon
	g_caliLinkEncoder :ARRAY[1..g_sArmNum, 1..g_setupJntNum] OF DINT :=
		[3511708, 21210622, 1977753, 9295000, 9311970,
		  11205276, 16093586, 3084321, 783598, 13445092,
		 844948, 14389054, 878439, 13364040, 5122582,
		  14940512, 22936561, 4169014, 13457164, 13393096];
	
	 // if absolute encoder value cross zeros within joint motion range
	g_linkEncZeroCross :ARRAY[1..g_sArmNum, 1..g_setupJntNum] OF INT :=
		[0, 0, 0, 1, 0,
		 0, 0, 0, 1, 1,
		 1, 0, 0, 1, 0,
		 1, 0, 0, 1, 1];
		 
//################ DO NOT modify parameters below ###########################
	// abolute encoder expanded limit buffer in case there is calibrtion error at limit position
	g_linkEncLimitBuffer : DINT := 100000;

	// absolute encoder direction
	g_asbEncoderDir :ARRAY[1..g_setupJntNum] OF INT :=[-1, -1, -1, 1, -1];
													
	// flag if joint can rotate multiple cycles
	g_multipleCyclesJoint :ARRAY[1..g_sArmNum, 1..g_setupJntNum] OF INT :=
		[0, 0, 0, 0, 0,
		 0, 0, 0, 0, 0,
		 0, 0, 0, 0, 0,
		 0, 0, 0, 0, 0];
		 
	// joint position at link encoder calibrated point
	g_linkEncCaliJntPos :ARRAY[1..g_sArmNum, 1..g_setupJntNum] OF LREAL :=
		[-140*g_deg2Rad, 0.779, 0.0, 90.0*g_deg2Rad, 0.0,
		 -115*g_deg2Rad, 0.607, 0.0, 90.0*g_deg2Rad, 0.0,
		 -65*g_deg2Rad, 0.607, 0.0, 90.0*g_deg2Rad, 0.0,
 		 -40*g_deg2Rad, 0.779, 0.0, 90.0*g_deg2Rad, 0.0];
	
END_VAR

// ---- GVLs/SetupArms/GVL_SetupMotorParameters.TcGVL
{attribute 'global_init_slot' := '49991'}
{attribute 'qualified_only'}
VAR_GLOBAL CONSTANT
	// encoder resolution
	//TODO: resolution of joint 2/3 need verification
	g_incEncoderRes :ARRAY[1..g_setupJntNum] OF DINT :=[5(65536)];
	g_absEncoderRes :ARRAY[1..g_setupJntNum] OF DINT :=[16777216,8192, 8192, 2(16777216)];
	
	// reduction ratio
	g_motorReduction :ARRAY[1..g_setupJntNum] OF LREAL :=[1,1,2*pi/0.020,81,161];
	g_absEncoderReduction :ARRAY[1..g_setupJntNum] OF LREAL :=[1.0, 2*pi/0.002 , 2*PI/0.002, 1.0, 1.0];
	
	// motor parameters
	g_motorTrqConst :ARRAY[1..g_setupJntNum] OF LREAL :=[ 1,1,0.16,0.1,0.16];
	g_motorMaxCurrent :ARRAY[1..g_setupJntNum] OF LREAL :=[ 1,1,5600,3800,5600];//mA
	
	// motor and absEncoder direction
	g_motorDir :ARRAY[1..g_setupJntNum] OF INT :=[-1, -1, 1, -1, 1];
																												 
	// joint position limit
	g_minJntPos: ARRAY[1..g_sArmNum,  1..g_setupJntNum] OF LREAL:=[ (-140-50)*g_deg2Rad, 0.779-0.36,0.00,-1.2351,-1.7473,
																	(-115-50)*g_deg2Rad, 0.607-0.36,0.00,-1.2351,-1.7473,
																	(-65-50)*g_deg2Rad, 0.607-0.36,0.00,-1.2351,-1.7473,
																	(-40-50)*g_deg2Rad, 0.779-0.36,0.00,-1.2351,-1.7473];	
	g_maxJntPos: ARRAY[1..g_sArmNum,  1..g_setupJntNum] OF LREAL:=[ (-140+50)*g_deg2Rad, 0.779,0.200,4.5579,1.7284,
																	(-115+50)*g_deg2Rad, 0.607,0.200,4.5579,1.7284,
																	(-65+50)*g_deg2Rad, 0.607,0.200,4.5579,1.7284,
																	(-40+50)*g_deg2Rad, 0.779,0.200,4.5579,1.7284];	
	
	// joint velocity limit
	g_maxJntVel :ARRAY[1..g_setupJntNum] OF LREAL :=[0.1, 0.1, 0.1, 0.1, 0.1];
	
END_VAR

// ---- GVLs/SetupArms/GVL_SetupArmKinematic.TcGVL
// use slot attribute larger than 49990, which is the default one, if it depends on variable in other file
{attribute 'global_init_slot' := '49991'} 
{attribute 'qualified_only'}
VAR_GLOBAL CONSTANT 

(* 
% setup arm
% 1        0      0   q1      0
% 2        90     a2   0      q2
% 3        -90     0   0       q3
% 4        0       0   q4      d4
% 5        -90      0   q5      0
*)
g_setupA2:ARRAY[1..4] OF LREAL:=[0.019,0.136, 0.136, 0.1825 ];
g_setupD4:ARRAY[1..4] OF LREAL:=[0.5205,0.3545, 0.3545, 0.5205 ];
g_L :LREAL:= 0.3;// need to be replace by real instrument parameters;
g_a : LREAL :=0.01;// need to be replace by real instrument parameters;
g_b :LREAL :=0;// need to be replace by real instrument parameters;

//alpha,a,d,theta	
g_setupArmDH:ARRAY[1..5,1..4] OF LREAL  :=[   0,   0,   0,     0,
											PI/2,  g_setupA2[1],   0,      0,
											-PI/2,  0,   0,       0,
											0,       0,   0,      g_setupA2[2],
											-PI/2,   0,   0,      0];


END_VAR

// ---- GVLs/SetupArms/GVL_SetupControlParameters.TcGVL
{attribute 'global_init_slot' := '49991'}
{attribute 'qualified_only'}
VAR_GLOBAL CONSTANT
	// filter cut-off frequency for velocity and torque
	g_curJntVelLpfCutoffFreq :LREAL := 30;
	g_cmdJntTrqLpfCutoffFreq :LREAL := 300;
	g_curJntTrqLpfCutoffFreq :LREAL := 300;
	
	// setup arm joint position controller parameters
	g_posKp :ARRAY[1..g_setupJntNum] OF LREAL :=[0.0, 0.0, 0.0, 0.0, 2000];
	g_posKd :ARRAY[1..g_setupJntNum] OF LREAL :=[0.0, 0.0, 0.0, 0.0, 200 ];
	g_posKi :ARRAY[1..g_setupJntNum] OF LREAL :=[0.0, 0.0, 0.0, 0.0, 5000];
	g_posKiLimit :ARRAY[1..g_setupJntNum] OF LREAL :=[0.0, 0.0, 0.0, 0.0, 2000];// define in current
	g_posCtrlLimit :ARRAY[1..g_setupJntNum] OF LREAL :=[0.0, 0.0, 0.0, 0.0, 5000];// define in current
	
END_VAR

// ---- GVLs/SlaveArms/GVL_SlaveArmDynamics.TcGVL
{attribute 'global_init_slot' := '49992'}
{attribute 'qualified_only'}
// Robot3 --dynamic parameters of slave arms
VAR_GLOBAL CONSTANT
	
	// arm gravity parameters
(*graParam=[ 9.8*m5,...
           0.41601*m2 + 0.41601*m3 + 0.0000216012*m4 + 0.0000216012*m5 + 9.8*mx1 - 1.3639*mx3 - 9.70463*my3,...
           9.8*mz2 - 9.8*my5 - 9.8*my1 + 9.8*mz3 + 9.8*mz4,...
           2.19651*m3 + 2.19651*m4 + 0.00000258969*m5 + 8.64766*mx2 - 4.61063*my2 + 9.8*my4 + 9.8*mz5,...
          1.1711*m3 + 1.1711*m4 + 0.00000122416*m5 + 4.61063*mx2 - 9.8*mx4 - 9.8*mx5 + 8.64766*my2]'
*)				
	// robot No.4
	g_gravityParam :ARRAY[1..4,1..5] OF REAL := 
	[ 7.5951,    1.6336,   -4.2417,    9.4106,    4.7289,
	  7.4741,    3.7472,   -4.4567,   10.5517,    7.6095,
	  7.6732,    3.7472,   -4.4458,    9.6721,    7.2742,
	  7.4582,    3.5688,   -3.7215,    9.2746,    5.7641];
	 
	g_gravityTrocar :ARRAY[1..5] OF REAL :=[0.1661, -0.4124,  0.0964,   -0.7987,   -0.6999 ];
	g_gravityInstrument :ARRAY[1..5] OF REAL :=[ 3.1217,  -0.3099,   0.0778,   -1.2498,   -0.8041];
	g_gravityEndoscope :ARRAY[1..5] OF REAL :=[10.8619,  -0.8575,   -1.0274,   -0.2425,   -0.0869];
	
	// joint friction(with instrument mounted)
	g_slaveJntFriction :ARRAY[1..g_sArmNum, 1..g_sJntNum] OF LREAL :=
			[ 5.3354,    9.5437,    4.6271,  0.03, 0.03, 0.03, 0.03, 0,
			  4.5927,    9.6040,    3.7367, 0.03, 0.03, 0.03, 0,
		      4.3557,    8.4286,    5.9078,  0.03, 0.03, 0.03, 0.03, 0,
              4.1447,    7.2202,    6.8253,  0.03, 0.03, 0.03, 0.03, 0	 ];
			  
	//################ DO NOT modify parameters below ###########################
	//################ dynamic reference model parameters below ###########################
	// link mass [m1, m2, m3, m4, m5]
	g_linkMass :ARRAY[1..5] OF LREAL :=[5.6565, 1.4613, 1.149, 1.5362, 0.6679] ;
	
	// lin center of amss
	g_linkCOM :ARRAY[1..5,1..3] OF LREAL :=  [ 0.0566,    0.0302,   -0.4685,
											   0.1191,   -0.0011,   -0.0588,
											   0.1238,    0.0003,   -0.0120,
											   0.0427,    0.0924,   -0.0004,
											   -0.0262,        0,   -0.0292];
	// link  inertial
    // [Ixx,Iyy,Izz, Ixy,Ixz, Iyz]
 	g_linkInertia :ARRAY[1..5,1..6] OF LREAL :=[0.0735,    0.0738,    0.0144,    0.0016,   -0.0000,   -0.0079,
												0.0016,    0.0190,    0.0185,         0,    0.0027,         0,
											   0.0009,    0.0167,    0.0166,         0,    0.0012,         0,
												0.0009,    0.0167,    0.0166,         0,    0.0012,         0,
											  0.0009,    0.0167,    0.0166,         0,    0.0012,         0];

	
	//  motor inertial at link size
	g_motorInertia :ARRAY[1..3] OF LREAL := [0.00004487, 0.00004487, 0.0000002280];

END_VAR

// ---- GVLs/SlaveArms/GVL_SlaveArmKinematic.TcGVL
// use slot attribute larger than 49990, which is the default one, if it depends on variable in other file
{attribute 'global_init_slot' := '49991'} 
{attribute 'qualified_only'}
VAR_GLOBAL CONSTANT 

(* 
% paramters definiton:
% d1: distance from joint1 to remote center
% L: instrument length
% a: distance from joint5 to joint 6 on tool
% b: distantce form joint 6 to tcp on tool
% DH definition:
% index    alpha   a   theta   d
% 1        90      0   q1      d1
% 2        -90     0   q2      0
% 3        -90     0   0       q3
% 4        0       0   q4      -L
% 5        90      0   q5      0
% 6        90      a   q6      0
% 7      0       b   0       0

*)
g_d1:LREAL:=0.8046229;
g_L :LREAL:= 0.3;// need to be replace by real instrument parameters;
g_a : LREAL :=0.01;// need to be replace by real instrument parameters;
g_b :LREAL :=0;// need to be replace by real instrument parameters;

//alpha,a,d,theta	
g_slaveArmDH:ARRAY[1..7,1..4] OF LREAL :=[PI/2,	0,		g_d1,	0,      
											-pi/2,	0,		0,		0,
											-PI/2,	0,		0,		0,
									        0,		0,		-g_L,	0,       
											pi/2,	0,		0,		0,
								            pi/2,	g_a,	0,		0,
							         		0,		g_b, 	0,		0];
			

//%% DH definetion
//% paramters definiton:
//% a: distance from joint5 to joint 6 on tool
//% b: distantce form joint 6 to tcp on tool
//% DH definition:
//% index    alpha   a        theta           d
//% 1        90      0        J1+180          0
//% 2        90     42.45     J2-61.935       0
//% P1       0      254       -J2-200.065     0
//% P2       0      305       J2+82              0
//% 3        -90     119.5    0               J3-224.133
//% 4        0       0        J4              -L
//% 5        90      0        J5              0
//% 6        90      a        J6              0
//% tcp      0       b        0               0
g_slaveArmFullDH:ARRAY[1..9,1..4] OF LREAL :=[ PI/2,   	0,   		PI,      			502.591/1000,
												PI/2,  	42.45/1000,	-61.935*g_deg2rad,      0,
												0,      254.0/1000,   -200.065*g_deg2rad,       0,
												0,   	305.0/1000,   82.0*g_deg2rad,             0,
												-PI/2,  119.5/1000, 0,       			-224.133/1000,
												0,      0,   		0,	      			-g_L,
												PI/2,   0,   		0,      			0,
												PI/2,   g_a,   		0,      			0,
												0,       g_b,   	0,      			0];

						
g_slaveArmDHErr:ARRAY[1..4,1..13] OF LREAL :=[ -0.0251,    0.0032,    0.0200,    -0.0064,   -0.0039,    0.0101,   -0.0153,   -0.0117,   -0.0586,   -0.0021,    0.036,   -0.0058,   -0.0068,
											  0.0,	   -0.0084,    0.0179,      0.0,   -0.0195,   -0.0137,    0.0001,   -0.0154,   -0.0501,   -0.0033,    0.0379,   -0.0453,   -0.0019,
											  0.048,	-0.0085,	0.0106,	0.0068,	-0.0076,	-0.0169,	0.0067,	0.0222,	-0.0151,	0.0001,	0.0219,	-0.009,		-0.0065,
											  13(0)];

g_slaveArmBaseErr:ARRAY[1..4,1..2] OF LREAL :=[ -0.0064,    -0.0129,
											  0.0,	 0.0,
											  0.0056,	0.0038,
											  2(0)];
	
// rotation from joint7 to tcp
g_tcpRotation :Mat3d :=[0.0,	0.0,	1.0,
					    -1.0,	0.0,	0.0,
					    0.0,	-1.0,	0.0];

// minimum distance between instrument/endoscope tip and remote center
g_minInstruRCDis:LREAL := 0.03;
	
